C08974=1024.859,160.685,-112.460,168.492,47.875,158.974
C08975=1024.853,160.436,-112.438,168.489,47.879,158.974
C08976=1024.849,160.187,-112.416,168.486,47.884,158.975
C08977=1024.842,159.938,-112.393,168.482,47.888,158.975
C08978=1024.837,159.689,-112.372,168.480,47.892,158.976
C08979=1024.832,159.440,-112.349,168.476,47.897,158.976
C08980=1024.826,159.191,-112.328,168.472,47.901,158.977
C08981=1024.821,158.942,-112.306,168.470,47.905,158.977
C08982=1024.815,158.693,-112.285,168.466,47.910,158.978
C08983=1024.809,158.444,-112.263,168.464,47.914,158.978
C08984=1024.803,158.195,-112.241,168.460,47.918,158.978
C08985=1024.797,157.946,-112.220,168.456,47.923,158.979
C08986=1024.792,157.697,-112.198,168.454,47.928,158.979
C08987=1024.786,157.448,-112.177,168.450,47.932,158.980
C08988=1024.780,157.199,-112.155,168.446,47.937,158.980
C08989=1024.775,156.951,-112.134,168.444,47.941,158.981
C08990=1024.770,156.701,-112.112,168.440,47.946,158.981
C08991=1024.764,156.452,-112.091,168.438,47.950,158.982
C08992=1024.757,156.169,-112.066,168.433,47.955,158.982
C08993=1024.751,155.886,-112.042,168.430,47.960,158.983
C08994=1024.745,155.602,-112.017,168.426,47.965,158.983
C08995=1024.738,155.318,-111.992,168.423,47.970,158.984
C08996=1024.732,155.070,-111.971,168.419,47.974,158.984
C08997=1024.726,154.820,-111.950,168.416,47.979,158.985
C08998=1024.721,154.571,-111.929,168.414,47.984,158.985
C08999=1024.715,154.322,-111.907,168.410,47.988,158.985
C09000=1024.710,154.073,-111.885,168.407,47.992,158.986
C09001=1024.703,153.824,-111.864,168.404,47.997,158.986
C09002=1024.698,153.576,-111.843,168.401,48.001,158.987
C09003=1024.693,153.326,-111.822,168.397,48.006,158.987
C09004=1024.687,153.077,-111.800,168.394,48.010,158.988
C09005=1024.682,152.828,-111.779,168.391,48.015,158.988
C09006=1024.675,152.579,-111.757,168.388,48.019,158.989
C09007=1024.670,152.330,-111.736,168.385,48.023,158.989
C09008=1024.664,152.081,-111.715,168.382,48.028,158.990
C09009=1024.658,151.832,-111.693,168.378,48.033,158.990
C09010=1024.653,151.583,-111.673,168.375,48.037,158.990
C09011=1024.647,151.334,-111.651,168.372,48.042,158.991
C09012=1024.641,151.085,-111.630,168.369,48.046,158.992
C09013=1024.636,150.836,-111.609,168.366,48.051,158.992
C09014=1024.630,150.587,-111.588,168.363,48.055,158.992
C09015=1024.624,150.338,-111.566,168.360,48.059,158.993
C09016=1024.619,150.089,-111.546,168.356,48.064,158.993
C09017=1024.612,149.840,-111.524,168.354,48.069,158.994
C09018=1024.607,149.591,-111.503,168.350,48.073,158.994
C09019=1024.602,149.342,-111.482,168.347,48.077,158.995
C09020=1024.595,149.093,-111.460,168.344,48.082,158.995
C09021=1024.590,148.844,-111.440,168.341,48.087,158.996
C09022=1024.584,148.595,-111.418,168.338,48.091,158.996
C09023=1024.579,148.345,-111.398,168.335,48.095,158.997
C09024=1024.573,148.097,-111.376,168.332,48.100,158.997
C09025=1024.567,147.848,-111.355,168.329,48.105,158.998
C09026=1024.562,147.599,-111.334,168.325,48.109,158.998
C09027=1024.556,147.349,-111.313,168.322,48.113,158.998
C09028=1024.550,147.100,-111.292,168.319,48.118,158.999
C09029=1024.545,146.852,-111.271,168.316,48.123,158.999
C09030=1024.539,146.602,-111.250,168.313,48.127,159.000
C09031=1024.533,146.353,-111.229,168.310,48.131,159.000
C09032=1024.528,146.104,-111.208,168.307,48.136,159.001
C09033=1024.522,145.854,-111.187,168.304,48.141,159.001
C09034=1024.517,145.606,-111.166,168.301,48.145,159.002
C09035=1024.511,145.357,-111.145,168.298,48.150,159.002
C09036=1024.505,145.108,-111.124,168.295,48.155,159.003
C09037=1024.499,144.859,-111.104,168.291,48.159,159.003
C09038=1024.494,144.610,-111.083,168.289,48.163,159.004
C09039=1024.488,144.360,-111.062,168.285,48.168,159.004
C09040=1024.483,144.111,-111.041,168.282,48.173,159.005
C09041=1024.477,143.863,-111.021,168.280,48.177,159.005
C09042=1024.470,143.613,-110.999,168.276,48.182,159.006
C09043=1024.465,143.364,-110.979,168.274,48.187,159.006
C09044=1024.460,143.115,-110.958,168.270,48.191,159.006
C09045=1024.453,142.866,-110.937,168.267,48.195,159.007
C09046=1024.448,142.617,-110.917,168.264,48.200,159.008
C09047=1024.443,142.368,-110.896,168.261,48.205,159.008
C09048=1024.437,142.119,-110.875,168.258,48.209,159.009
C09049=1024.430,141.870,-110.855,168.255,48.214,159.009
C09050=1024.425,141.621,-110.834,168.252,48.219,159.010
C09051=1024.420,141.372,-110.813,168.249,48.222,159.010
C09052=1024.414,141.122,-110.792,168.246,48.227,159.010
C09053=1024.408,140.873,-110.771,168.243,48.232,159.011
C09054=1024.402,140.625,-110.751,168.240,48.237,159.011
C09055=1024.397,140.375,-110.731,168.237,48.241,159.012
C09056=1024.391,140.091,-110.707,168.234,48.246,159.012
C09057=1024.384,139.808,-110.683,168.231,48.251,159.013
C09058=1024.378,139.524,-110.659,168.226,48.257,159.013
C09059=1024.371,139.241,-110.636,168.223,48.262,159.014
C09060=1024.366,138.992,-110.616,168.221,48.267,159.015
C09061=1024.360,138.743,-110.595,168.217,48.271,159.015
C09062=1024.354,138.493,-110.574,168.214,48.275,159.015
C09063=1024.348,138.244,-110.554,168.211,48.280,159.016
C09064=1024.343,137.995,-110.534,168.208,48.285,159.017
C09065=1024.338,137.746,-110.513,168.205,48.289,159.017
C09066=1024.331,137.496,-110.493,168.202,48.294,159.018
C09067=1024.326,137.248,-110.471,168.199,48.299,159.018
C09068=1024.320,136.999,-110.451,168.197,48.303,159.019
C09069=1024.315,136.750,-110.431,168.193,48.308,159.019
C09070=1024.309,136.501,-110.410,168.191,48.313,159.020
C09071=1024.303,136.251,-110.390,168.188,48.316,159.020
C09072=1024.297,136.002,-110.369,168.184,48.321,159.020
C09073=1024.291,135.753,-110.349,168.182,48.326,159.021
C09074=1024.286,135.504,-110.329,168.178,48.331,159.021
C09075=1024.280,135.255,-110.309,168.176,48.335,159.022
C09076=1024.274,135.005,-110.288,168.173,48.340,159.022
C09077=1024.268,134.757,-110.268,168.170,48.345,159.023
C09078=1024.263,134.508,-110.248,168.167,48.349,159.023
C09079=1024.257,134.259,-110.228,168.164,48.354,159.024
C09080=1024.252,134.010,-110.207,168.161,48.359,159.024
C09081=1024.246,133.761,-110.187,168.158,48.363,159.025
C09082=1024.241,133.512,-110.167,168.155,48.368,159.025
C09083=1024.234,133.262,-110.147,168.152,48.373,159.026
C09084=1024.229,133.012,-110.126,168.149,48.377,159.026
C09085=1024.223,132.764,-110.106,168.146,48.382,159.027
C09086=1024.218,132.514,-110.086,168.143,48.386,159.027
C09087=1024.212,132.266,-110.066,168.140,48.391,159.028
C09088=1024.207,132.017,-110.045,168.138,48.395,159.028
C09089=1024.201,131.768,-110.025,168.134,48.400,159.029
C09090=1024.195,131.518,-110.004,168.132,48.405,159.029
C09091=1024.189,131.269,-109.984,168.128,48.409,159.030
C09092=1024.183,131.020,-109.964,168.126,48.414,159.030
C09093=1024.178,130.771,-109.945,168.123,48.419,159.031
C09094=1024.173,130.521,-109.924,168.120,48.423,159.031
C09095=1024.167,130.273,-109.904,168.117,48.428,159.032
C09096=1024.161,130.023,-109.884,168.114,48.433,159.032
C09097=1024.155,129.775,-109.864,168.112,48.437,159.033
C09098=1024.150,129.525,-109.844,168.108,48.442,159.033
C09099=1024.144,129.276,-109.824,168.105,48.447,159.034
C09100=1024.137,129.027,-109.804,168.102,48.452,159.034
C09101=1024.131,128.777,-109.785,168.099,48.456,159.035
C09102=1024.126,128.528,-109.764,168.097,48.461,159.035
C09103=1024.120,128.280,-109.744,168.094,48.465,159.036
C09104=1024.114,128.030,-109.725,168.091,48.470,159.036
C09105=1024.108,127.781,-109.705,168.088,48.475,159.037
C09106=1024.102,127.532,-109.685,168.085,48.480,159.037
C09107=1024.097,127.283,-109.666,168.083,48.485,159.038
C09108=1024.091,127.034,-109.646,168.079,48.490,159.039
C09109=1024.086,126.784,-109.626,168.077,48.494,159.039
C09110=1024.080,126.536,-109.606,168.073,48.499,159.040
C09111=1024.073,126.286,-109.586,168.071,48.504,159.040
C09112=1024.067,126.037,-109.567,168.067,48.509,159.041
C09113=1024.061,125.788,-109.547,168.065,48.513,159.041
C09114=1024.056,125.538,-109.527,168.062,48.518,159.042
C09115=1024.051,125.289,-109.507,168.059,48.523,159.042
C09116=1024.045,125.041,-109.487,168.056,48.527,159.043
C09117=1024.039,124.791,-109.468,168.053,48.532,159.043
C09118=1024.033,124.542,-109.448,168.050,48.537,159.044
C09119=1024.027,124.293,-109.428,168.047,48.541,159.044
C09120=1024.021,124.009,-109.406,168.044,48.547,159.045
C09121=1024.014,123.726,-109.384,168.041,48.552,159.046
C09122=1024.008,123.442,-109.361,168.038,48.557,159.046
C09123=1024.002,123.158,-109.339,168.035,48.563,159.047
C09124=1023.996,122.909,-109.319,168.031,48.568,159.047
C09125=1023.990,122.660,-109.299,168.029,48.572,159.048
C09126=1023.984,122.411,-109.279,168.026,48.577,159.048
C09127=1023.978,122.161,-109.260,168.023,48.582,159.049
C09128=1023.972,121.913,-109.240,168.020,48.586,159.049
C09129=1023.967,121.663,-109.221,168.017,48.591,159.050
C09130=1023.961,121.414,-109.200,168.014,48.596,159.050
C09131=1023.956,121.165,-109.181,168.012,48.600,159.051
C09132=1023.950,120.916,-109.161,168.009,48.605,159.051
C09133=1023.944,120.666,-109.142,168.006,48.610,159.052
C09134=1023.938,120.417,-109.123,168.003,48.614,159.052
C09135=1023.932,120.168,-109.103,168.000,48.619,159.053
C09136=1023.927,119.919,-109.084,167.998,48.624,159.053
C09137=1023.921,119.670,-109.063,167.994,48.629,159.054
C09138=1023.916,119.420,-109.044,167.992,48.633,159.054
C09139=1023.910,119.171,-109.024,167.989,48.638,159.055
C09140=1023.904,118.922,-109.005,167.986,48.643,159.055
C09141=1023.898,118.672,-108.985,167.984,48.647,159.056
C09142=1023.892,118.424,-108.965,167.980,48.652,159.056
C09143=1023.887,118.175,-108.946,167.978,48.657,159.057
C09144=1023.882,117.926,-108.927,167.976,48.661,159.057
C09145=1023.876,117.676,-108.907,167.972,48.666,159.058
C09146=1023.871,117.427,-108.887,167.970,48.671,159.058
C09147=1023.865,117.178,-108.867,167.966,48.675,159.059
C09148=1023.859,116.929,-108.848,167.964,48.680,159.059
C09149=1023.853,116.679,-108.829,167.961,48.685,159.060
C09150=1023.847,116.430,-108.809,167.958,48.689,159.060
C09151=1023.842,116.182,-108.790,167.956,48.694,159.061
C09152=1023.837,115.932,-108.771,167.953,48.699,159.062
C09153=1023.831,115.683,-108.750,167.950,48.703,159.062
C09154=1023.826,115.434,-108.731,167.947,48.708,159.063
C09155=1023.820,115.184,-108.712,167.945,48.713,159.063
C09156=1023.814,114.935,-108.693,167.941,48.718,159.064
C09157=1023.808,114.686,-108.673,167.939,48.722,159.064
C09158=1023.803,114.437,-108.654,167.936,48.726,159.064
C09159=1023.797,114.188,-108.635,167.933,48.731,159.065
C09160=1023.791,113.939,-108.615,167.930,48.735,159.065
C09161=1023.786,113.690,-108.595,167.928,48.740,159.066
C09162=1023.781,113.440,-108.575,167.925,48.745,159.066
C09163=1023.775,113.190,-108.556,167.922,48.750,159.067
C09164=1023.770,112.942,-108.537,167.920,48.754,159.067
C09165=1023.764,112.693,-108.517,167.917,48.759,159.068
C09166=1023.758,112.443,-108.498,167.914,48.764,159.068
C09167=1023.753,112.194,-108.479,167.912,48.768,159.069
C09168=1023.746,111.945,-108.460,167.908,48.773,159.069
C09169=1023.741,111.695,-108.441,167.906,48.778,159.070
C09170=1023.735,111.447,-108.422,167.903,48.782,159.071
C09171=1023.730,111.197,-108.403,167.900,48.787,159.071
C09172=1023.724,110.948,-108.384,167.897,48.792,159.072
C09173=1023.718,110.698,-108.364,167.895,48.796,159.072
C09174=1023.712,110.450,-108.345,167.892,48.801,159.073
C09175=1023.707,110.201,-108.326,167.889,48.806,159.073
C09176=1023.701,109.952,-108.307,167.886,48.811,159.074
C09177=1023.695,109.702,-108.288,167.884,48.816,159.074
C09178=1023.689,109.453,-108.268,167.881,48.821,159.075
C09179=1023.683,109.204,-108.250,167.878,48.825,159.075
C09180=1023.678,108.954,-108.231,167.876,48.830,159.076
C09181=1023.673,108.705,-108.212,167.873,48.835,159.076
C09182=1023.666,108.456,-108.194,167.870,48.840,159.077
C09183=1023.660,108.206,-108.175,167.867,48.844,159.077
C09184=1023.653,107.923,-108.153,167.864,48.850,159.078
C09185=1023.647,107.639,-108.131,167.861,48.855,159.079
C09186=1023.641,107.355,-108.110,167.858,48.861,159.079
C09187=1023.634,107.071,-108.089,167.855,48.866,159.080
C09188=1023.629,106.822,-108.070,167.852,48.871,159.080
C09189=1023.622,106.573,-108.051,167.849,48.876,159.081
C09190=1023.617,106.323,-108.032,167.847,48.881,159.081
C09191=1023.611,106.074,-108.013,167.843,48.885,159.082
C09192=1023.605,105.825,-107.994,167.841,48.890,159.082
C09193=1023.599,105.576,-107.975,167.839,48.895,159.083
C09194=1023.594,105.327,-107.956,167.835,48.900,159.083
C09195=1023.588,105.078,-107.938,167.833,48.904,159.084
C09196=1023.582,104.828,-107.919,167.830,48.910,159.085
C09197=1023.577,104.579,-107.900,167.827,48.914,159.085
C09198=1023.570,104.330,-107.881,167.825,48.919,159.086
C09199=1023.565,104.081,-107.862,167.821,48.924,159.086
C09200=1023.559,103.832,-107.844,167.819,48.928,159.087
C09201=1023.553,103.582,-107.825,167.817,48.933,159.087
C09202=1023.548,103.333,-107.806,167.813,48.938,159.088
C09203=1023.542,103.084,-107.787,167.811,48.943,159.088
C09204=1023.536,102.834,-107.768,167.809,48.947,159.089
C09205=1023.531,102.585,-107.749,167.805,48.952,159.089
C09206=1023.525,102.336,-107.731,167.803,48.957,159.090
C09207=1023.519,102.086,-107.712,167.800,48.961,159.090
C09208=1023.513,101.837,-107.694,167.797,48.966,159.091
C09209=1023.508,101.589,-107.675,167.795,48.971,159.091
C09210=1023.502,101.339,-107.656,167.792,48.976,159.092
C09211=1023.496,101.089,-107.637,167.790,48.980,159.092
C09212=1023.491,100.841,-107.619,167.786,48.985,159.093
C09213=1023.485,100.591,-107.599,167.784,48.990,159.093
C09214=1023.480,100.342,-107.582,167.782,48.994,159.094
C09215=1023.474,100.093,-107.563,167.778,48.999,159.094
C09216=1023.468,99.844,-107.544,167.776,49.004,159.095
C09217=1023.462,99.594,-107.525,167.773,49.008,159.095
C09218=1023.457,99.345,-107.507,167.770,49.014,159.096
C09219=1023.451,99.096,-107.488,167.768,49.019,159.097
C09220=1023.445,98.847,-107.470,167.766,49.023,159.097
C09221=1023.440,98.597,-107.451,167.762,49.028,159.098
C09222=1023.433,98.348,-107.433,167.760,49.033,159.098
C09223=1023.428,98.099,-107.415,167.756,49.038,159.099
C09224=1023.422,97.849,-107.396,167.754,49.043,159.099
C09225=1023.416,97.600,-107.378,167.752,49.048,159.100
C09226=1023.410,97.352,-107.359,167.749,49.053,159.100
C09227=1023.405,97.102,-107.341,167.746,49.057,159.101
C09228=1023.398,96.852,-107.322,167.744,49.062,159.101
C09229=1023.393,96.603,-107.305,167.740,49.067,159.102
C09230=1023.387,96.354,-107.285,167.738,49.071,159.102
C09231=1023.381,96.105,-107.268,167.736,49.077,159.103
C09232=1023.375,95.856,-107.249,167.733,49.082,159.104
C09233=1023.370,95.606,-107.231,167.730,49.086,159.104
C09234=1023.364,95.357,-107.212,167.728,49.091,159.105
C09235=1023.358,95.108,-107.194,167.724,49.096,159.105
C09236=1023.353,94.859,-107.176,167.722,49.100,159.106
C09237=1023.346,94.609,-107.158,167.720,49.105,159.106
C09238=1023.340,94.360,-107.139,167.716,49.110,159.107
C09239=1023.335,94.111,-107.121,167.714,49.115,159.107
C09240=1023.329,93.861,-107.103,167.712,49.120,159.108
C09241=1023.323,93.612,-107.085,167.709,49.125,159.108
C09242=1023.318,93.362,-107.066,167.706,49.130,159.109
C09243=1023.312,93.114,-107.048,167.704,49.134,159.109
C09244=1023.306,92.864,-107.030,167.700,49.139,159.110
C09245=1023.301,92.616,-107.011,167.698,49.144,159.110
C09246=1023.295,92.366,-106.993,167.696,49.148,159.111
C09247=1023.289,92.116,-106.975,167.692,49.153,159.111
C09248=1023.282,91.833,-106.954,167.690,49.159,159.112
C09249=1023.276,91.548,-106.933,167.687,49.164,159.113
C09250=1023.270,91.265,-106.912,167.684,49.169,159.113
C09251=1023.263,90.981,-106.892,167.681,49.175,159.114
C09252=1023.257,90.732,-106.874,167.678,49.179,159.114
C09253=1023.252,90.482,-106.855,167.675,49.184,159.115
C09254=1023.246,90.234,-106.837,167.673,49.189,159.115
C09255=1023.240,89.984,-106.819,167.670,49.194,159.116
C09256=1023.235,89.735,-106.801,167.667,49.199,159.116
C09257=1023.229,89.486,-106.782,167.664,49.203,159.117
C09258=1023.223,89.236,-106.764,167.662,49.208,159.117
C09259=1023.217,88.987,-106.747,167.659,49.214,159.118
C09260=1023.211,88.738,-106.729,167.657,49.218,159.118
C09261=1023.205,88.488,-106.711,167.654,49.223,159.119
C09262=1023.199,88.240,-106.693,167.651,49.228,159.119
C09263=1023.193,87.990,-106.675,167.649,49.232,159.120
C09264=1023.188,87.741,-106.657,167.647,49.238,159.121
C09265=1023.182,87.491,-106.639,167.643,49.243,159.121
C09266=1023.176,87.242,-106.622,167.641,49.247,159.122
C09267=1023.170,86.992,-106.604,167.638,49.252,159.122
C09268=1023.164,86.744,-106.586,167.635,49.257,159.123
C09269=1023.158,86.494,-106.568,167.633,49.262,159.123
C09270=1023.153,86.245,-106.550,167.631,49.267,159.124
C09271=1023.147,85.995,-106.532,167.627,49.272,159.124
C09272=1023.141,85.746,-106.515,167.625,49.277,159.125
C09273=1023.135,85.497,-106.497,167.623,49.281,159.125
C09274=1023.129,85.247,-106.479,167.619,49.286,159.126
C09275=1023.123,84.998,-106.461,167.617,49.291,159.126
C09276=1023.117,84.749,-106.443,167.615,49.296,159.127
C09277=1023.111,84.500,-106.425,167.612,49.301,159.128
C09278=1023.106,84.251,-106.407,167.609,49.306,159.128
C09279=1023.100,84.002,-106.390,167.607,49.310,159.129
C09280=1023.094,83.752,-106.372,167.603,49.315,159.129
C09281=1023.089,83.503,-106.354,167.601,49.320,159.130
C09282=1023.083,83.253,-106.336,167.599,49.325,159.130
C09283=1023.077,83.004,-106.319,167.595,49.330,159.131
C09284=1023.072,82.754,-106.300,167.593,49.335,159.131
C09285=1023.066,82.505,-106.283,167.591,49.340,159.132
C09286=1023.061,82.256,-106.265,167.588,49.345,159.132
C09287=1023.054,82.006,-106.247,167.585,49.349,159.133
C09288=1023.049,81.757,-106.230,167.583,49.354,159.133
C09289=1023.043,81.507,-106.212,167.580,49.359,159.134
C09290=1023.037,81.258,-106.194,167.577,49.364,159.134
C09291=1023.032,81.009,-106.177,167.575,49.368,159.135
C09292=1023.026,80.759,-106.159,167.573,49.373,159.135
C09293=1023.020,80.510,-106.141,167.569,49.378,159.136
C09294=1023.015,80.261,-106.123,167.567,49.382,159.136
C09295=1023.008,80.012,-106.106,167.564,49.387,159.137
C09296=1023.002,79.763,-106.089,167.561,49.392,159.137
C09297=1022.997,79.514,-106.071,167.559,49.397,159.138
C09298=1022.991,79.264,-106.053,167.557,49.402,159.139
C09299=1022.985,79.015,-106.036,167.554,49.407,159.139
C09300=1022.979,78.765,-106.018,167.551,49.412,159.140
C09301=1022.973,78.516,-106.000,167.549,49.416,159.140
C09302=1022.968,78.267,-105.982,167.546,49.421,159.141
C09303=1022.962,78.018,-105.965,167.543,49.426,159.141
C09304=1022.956,77.768,-105.947,167.541,49.431,159.142
C09305=1022.951,77.519,-105.929,167.538,49.435,159.142
C09306=1022.945,77.270,-105.911,167.536,49.440,159.143
C09307=1022.939,77.020,-105.895,167.533,49.445,159.143
C09308=1022.934,76.771,-105.877,167.530,49.450,159.144
C09309=1022.928,76.521,-105.859,167.528,49.454,159.144
C09310=1022.922,76.272,-105.842,167.525,49.459,159.145
C09311=1022.916,76.023,-105.825,167.522,49.464,159.145
C09312=1022.909,75.739,-105.804,167.519,49.470,159.146
C09313=1022.903,75.455,-105.785,167.516,49.475,159.146
C09314=1022.896,75.171,-105.765,167.513,49.481,159.147
C09315=1022.890,74.888,-105.746,167.510,49.487,159.148
C09316=1022.884,74.638,-105.728,167.508,49.491,159.148
C09317=1022.878,74.388,-105.711,167.505,49.496,159.149
C09318=1022.872,74.140,-105.694,167.502,49.501,159.149
C09319=1022.867,73.891,-105.676,167.500,49.506,159.150
C09320=1022.860,73.641,-105.658,167.498,49.511,159.151
C09321=1022.854,73.392,-105.642,167.494,49.516,159.151
C09322=1022.849,73.143,-105.625,167.492,49.521,159.151
C09323=1022.843,72.893,-105.607,167.490,49.525,159.152
C09324=1022.837,72.644,-105.590,167.486,49.530,159.152
C09325=1022.831,72.394,-105.573,167.484,49.535,159.153
C09326=1022.826,72.145,-105.555,167.482,49.540,159.154
C09327=1022.820,71.895,-105.538,167.479,49.544,159.154
C09328=1022.814,71.646,-105.521,167.476,49.549,159.154
C09329=1022.808,71.397,-105.503,167.474,49.554,159.155
C09330=1022.803,71.148,-105.487,167.472,49.560,159.156
C09331=1022.796,70.898,-105.469,167.468,49.565,159.156
C09332=1022.791,70.649,-105.452,167.466,49.569,159.157
C09333=1022.785,70.400,-105.435,167.464,49.574,159.157
C09334=1022.779,70.151,-105.418,167.460,49.579,159.158
C09335=1022.773,69.900,-105.401,167.458,49.584,159.158
C09336=1022.768,69.651,-105.383,167.456,49.588,159.159
C09337=1022.762,69.403,-105.366,167.453,49.593,159.159
C09338=1022.756,69.153,-105.349,167.450,49.598,159.160
C09339=1022.750,68.903,-105.331,167.448,49.603,159.160
C09340=1022.744,68.654,-105.315,167.445,49.607,159.161
C09341=1022.739,68.405,-105.298,167.442,49.612,159.161
C09342=1022.733,68.156,-105.281,167.440,49.617,159.162
C09343=1022.727,67.906,-105.264,167.438,49.622,159.162
C09344=1022.722,67.656,-105.247,167.434,49.627,159.163
C09345=1022.715,67.407,-105.230,167.432,49.632,159.163
C09346=1022.710,67.158,-105.213,167.430,49.637,159.164
C09347=1022.704,66.909,-105.196,167.426,49.642,159.164
C09348=1022.699,66.659,-105.179,167.424,49.646,159.165
C09349=1022.692,66.410,-105.162,167.422,49.651,159.165
C09350=1022.686,66.160,-105.145,167.419,49.656,159.166
C09351=1022.680,65.912,-105.128,167.416,49.661,159.166
C09352=1022.675,65.662,-105.111,167.414,49.666,159.167
C09353=1022.669,65.413,-105.095,167.412,49.671,159.168
C09354=1022.663,65.163,-105.077,167.409,49.676,159.168
C09355=1022.657,64.913,-105.060,167.406,49.681,159.169
C09356=1022.651,64.664,-105.043,167.404,49.685,159.169
C09357=1022.646,64.415,-105.027,167.401,49.690,159.170
C09358=1022.640,64.166,-105.010,167.398,49.695,159.170
C09359=1022.634,63.917,-104.993,167.396,49.700,159.171
C09360=1022.628,63.667,-104.976,167.393,49.705,159.171
C09361=1022.622,63.418,-104.959,167.390,49.709,159.172
C09362=1022.616,63.168,-104.942,167.388,49.715,159.172
C09363=1022.611,62.919,-104.925,167.385,49.720,159.173
C09364=1022.605,62.669,-104.909,167.383,49.725,159.173
C09365=1022.598,62.420,-104.892,167.380,49.729,159.174
C09366=1022.592,62.170,-104.876,167.377,49.735,159.174
C09367=1022.586,61.921,-104.859,167.375,49.740,159.175
C09368=1022.580,61.672,-104.843,167.372,49.745,159.175
C09369=1022.575,61.422,-104.826,167.369,49.749,159.176
C09370=1022.569,61.173,-104.809,167.367,49.754,159.177
C09371=1022.563,60.924,-104.793,167.364,49.760,159.177
C09372=1022.556,60.674,-104.776,167.362,49.765,159.178
C09373=1022.550,60.425,-104.760,167.358,49.770,159.178
C09374=1022.544,60.175,-104.744,167.356,49.774,159.179
C09375=1022.539,59.926,-104.727,167.354,49.780,159.179
C09376=1022.532,59.642,-104.708,167.351,49.785,159.180
C09377=1022.525,59.358,-104.690,167.348,49.790,159.180
C09378=1022.519,59.074,-104.671,167.345,49.796,159.181
C09379=1022.512,58.790,-104.652,167.342,49.802,159.182
C09380=1022.506,58.541,-104.635,167.339,49.807,159.182
C09381=1022.500,58.292,-104.619,167.337,49.812,159.183
C09382=1022.494,58.042,-104.603,167.334,49.817,159.183
C09383=1022.488,57.792,-104.586,167.331,49.822,159.184
C09384=1022.482,57.543,-104.569,167.329,49.827,159.184
C09385=1022.476,57.293,-104.553,167.326,49.831,159.185
C09386=1022.470,57.045,-104.536,167.323,49.836,159.185
C09387=1022.464,56.795,-104.520,167.321,49.842,159.186
C09388=1022.458,56.546,-104.504,167.319,49.847,159.186
C09389=1022.452,56.296,-104.487,167.316,49.852,159.187
C09390=1022.447,56.047,-104.471,167.313,49.856,159.187
C09391=1022.441,55.797,-104.454,167.311,49.861,159.188
C09392=1022.435,55.548,-104.438,167.308,49.866,159.188
C09393=1022.429,55.299,-104.422,167.305,49.871,159.189
C09394=1022.423,55.049,-104.406,167.303,49.876,159.189
C09395=1022.417,54.800,-104.389,167.300,49.881,159.190
C09396=1022.412,54.550,-104.372,167.298,49.886,159.191
C09397=1022.406,54.301,-104.356,167.294,49.891,159.191
C09398=1022.400,54.052,-104.340,167.292,49.896,159.192
C09399=1022.394,53.802,-104.324,167.290,49.900,159.192
C09400=1022.388,53.553,-104.307,167.288,49.905,159.193
C09401=1022.382,53.304,-104.291,167.284,49.910,159.193
C09402=1022.376,53.054,-104.275,167.282,49.915,159.194
C09403=1022.371,52.805,-104.258,167.280,49.920,159.194
C09404=1022.365,52.555,-104.242,167.276,49.925,159.195
C09405=1022.359,52.306,-104.226,167.274,49.929,159.195
C09406=1022.353,52.057,-104.209,167.272,49.934,159.196
C09407=1022.347,51.807,-104.193,167.268,49.939,159.196
C09408=1022.341,51.558,-104.177,167.266,49.944,159.197
C09409=1022.335,51.309,-104.161,167.264,49.949,159.197
C09410=1022.329,51.059,-104.144,167.261,49.954,159.198
C09411=1022.324,50.810,-104.127,167.259,49.959,159.198
C09412=1022.318,50.560,-104.111,167.256,49.964,159.199
C09413=1022.312,50.311,-104.095,167.253,49.969,159.199
C09414=1022.306,50.062,-104.079,167.251,49.974,159.200
C09415=1022.301,49.812,-104.063,167.248,49.978,159.200
C09416=1022.295,49.562,-104.047,167.245,49.983,159.201
C09417=1022.289,49.313,-104.031,167.243,49.988,159.201
C09418=1022.283,49.064,-104.014,167.240,49.993,159.202
C09419=1022.277,48.814,-103.998,167.238,49.998,159.202
C09420=1022.272,48.565,-103.982,167.235,50.003,159.203
C09421=1022.266,48.316,-103.965,167.233,50.007,159.203
C09422=1022.260,48.067,-103.949,167.230,50.012,159.204
C09423=1022.254,47.817,-103.933,167.227,50.017,159.204
C09424=1022.249,47.567,-103.917,167.224,50.021,159.204
C09425=1022.243,47.318,-103.901,167.222,50.026,159.205
C09426=1022.237,47.068,-103.885,167.220,50.031,159.206
C09427=1022.232,46.819,-103.868,167.216,50.036,159.206
C09428=1022.226,46.569,-103.852,167.214,50.040,159.206
C09429=1022.220,46.320,-103.835,167.212,50.045,159.207
C09430=1022.215,46.071,-103.820,167.209,50.050,159.207
C09431=1022.209,45.822,-103.804,167.206,50.055,159.208
C09432=1022.203,45.572,-103.788,167.204,50.060,159.208
C09433=1022.197,45.323,-103.771,167.202,50.064,159.209
C09434=1022.191,45.073,-103.755,167.198,50.070,159.209
C09435=1022.186,44.823,-103.739,167.196,50.074,159.210
C09436=1022.180,44.574,-103.723,167.194,50.079,159.211
C09437=1022.175,44.325,-103.707,167.191,50.083,159.211
C09438=1022.169,44.076,-103.691,167.188,50.088,159.211
C09439=1022.163,43.826,-103.675,167.186,50.093,159.212
C09440=1022.156,43.542,-103.657,167.183,50.099,159.212
C09441=1022.150,43.258,-103.638,167.179,50.104,159.213
C09442=1022.143,42.974,-103.620,167.177,50.109,159.214
C09443=1022.136,42.689,-103.601,167.174,50.114,159.214
C09444=1022.131,42.440,-103.586,167.171,50.119,159.214
C09445=1022.125,42.191,-103.570,167.169,50.124,159.215
C09446=1022.120,41.941,-103.554,167.166,50.129,159.215
C09447=1022.114,41.692,-103.538,167.163,50.134,159.216
C09448=1022.108,41.442,-103.522,167.161,50.139,159.216
C09449=1022.101,41.192,-103.507,167.158,50.143,159.217
C09450=1022.096,40.944,-103.491,167.155,50.148,159.217
C09451=1022.090,40.694,-103.475,167.153,50.153,159.218
C09452=1022.084,40.445,-103.459,167.151,50.158,159.218
C09453=1022.079,40.195,-103.444,167.147,50.163,159.219
C09454=1022.073,39.945,-103.427,167.145,50.168,159.219
C09455=1022.067,39.697,-103.412,167.143,50.172,159.220
C09456=1022.061,39.447,-103.396,167.139,50.178,159.220
C09457=1022.055,39.198,-103.380,167.137,50.182,159.221
C09458=1022.049,38.948,-103.365,167.135,50.187,159.221
C09459=1022.043,38.698,-103.348,167.133,50.192,159.222
C09460=1022.038,38.449,-103.333,167.129,50.197,159.222
C09461=1022.032,38.200,-103.318,167.127,50.202,159.223
C09462=1022.026,37.950,-103.302,167.125,50.206,159.223
C09463=1022.020,37.701,-103.286,167.122,50.211,159.224
C09464=1022.015,37.451,-103.271,167.119,50.216,159.224
C09465=1022.009,37.202,-103.254,167.117,50.221,159.225
C09466=1022.003,36.952,-103.239,167.114,50.226,159.225
C09467=1021.997,36.702,-103.224,167.111,50.231,159.226
C09468=1021.991,36.453,-103.208,167.109,50.236,159.226
C09469=1021.985,36.204,-103.193,167.106,50.241,159.227
C09470=1021.979,35.955,-103.177,167.104,50.245,159.227
C09471=1021.974,35.705,-103.161,167.101,50.250,159.228
C09472=1021.967,35.455,-103.146,167.098,50.255,159.228
C09473=1021.962,35.206,-103.130,167.096,50.260,159.229
C09474=1021.956,34.957,-103.115,167.093,50.265,159.229
C09475=1021.950,34.707,-103.100,167.090,50.270,159.230
C09476=1021.944,34.457,-103.084,167.088,50.275,159.230
C09477=1021.938,34.209,-103.069,167.085,50.280,159.231
C09478=1021.933,33.959,-103.054,167.082,50.285,159.231
C09479=1021.926,33.709,-103.039,167.080,50.289,159.232
C09480=1021.921,33.460,-103.023,167.077,50.294,159.232
C09481=1021.915,33.211,-103.008,167.075,50.299,159.233
C09482=1021.909,32.961,-102.992,167.071,50.304,159.233
C09483=1021.903,32.711,-102.976,167.069,50.309,159.233
C09484=1021.897,32.462,-102.961,167.067,50.314,159.234
C09485=1021.892,32.212,-102.946,167.064,50.319,159.234
C09486=1021.885,31.963,-102.931,167.061,50.324,159.235
C09487=1021.880,31.714,-102.915,167.059,50.328,159.235
C09488=1021.873,31.464,-102.900,167.056,50.333,159.236
C09489=1021.868,31.214,-102.885,167.053,50.338,159.236
C09490=1021.863,30.965,-102.869,167.051,50.343,159.237
C09491=1021.856,30.716,-102.854,167.048,50.348,159.237
C09492=1021.850,30.466,-102.838,167.046,50.353,159.238
C09493=1021.845,30.217,-102.824,167.043,50.358,159.238
C09494=1021.839,29.967,-102.808,167.040,50.363,159.239
C09495=1021.833,29.718,-102.793,167.038,50.368,159.239
C09496=1021.828,29.468,-102.778,167.036,50.372,159.240
C09497=1021.821,29.219,-102.762,167.032,50.377,159.240
C09498=1021.816,28.970,-102.747,167.030,50.382,159.241
C09499=1021.810,28.720,-102.732,167.028,50.387,159.241
C09500=1021.804,28.470,-102.717,167.025,50.392,159.242
C09501=1021.799,28.221,-102.701,167.022,50.396,159.242
C09502=1021.792,27.971,-102.686,167.020,50.401,159.243
C09503=1021.786,27.722,-102.670,167.016,50.406,159.243
C09504=1021.777,27.319,-102.647,167.012,50.414,159.244
C09505=1021.768,26.917,-102.622,167.008,50.422,159.245
C09506=1021.758,26.513,-102.598,167.004,50.430,159.245
C09507=1021.748,26.111,-102.574,167.000,50.437,159.246
C09508=1021.743,25.861,-102.558,166.997,50.442,159.247
C09509=1021.737,25.612,-102.543,166.994,50.447,159.247
C09510=1021.731,25.362,-102.528,166.992,50.452,159.248
C09511=1021.725,25.113,-102.513,166.989,50.457,159.248
C09512=1021.719,24.864,-102.498,166.986,50.462,159.248
C09513=1021.713,24.614,-102.483,166.984,50.467,159.249
C09514=1021.708,24.365,-102.468,166.981,50.472,159.249
C09515=1021.701,24.115,-102.453,166.979,50.477,159.250
C09516=1021.693,23.735,-102.431,166.974,50.485,159.251
C09517=1021.684,23.354,-102.409,166.970,50.492,159.251
C09518=1021.674,22.974,-102.385,166.967,50.499,159.252
C09519=1021.666,22.594,-102.363,166.962,50.506,159.253
C09520=1021.660,22.344,-102.348,166.960,50.511,159.253
C09521=1021.654,22.095,-102.333,166.957,50.516,159.254
C09522=1021.648,21.845,-102.318,166.954,50.521,159.254
C09523=1021.642,21.596,-102.303,166.952,50.526,159.255
C09524=1021.637,21.346,-102.288,166.949,50.531,159.255
C09525=1021.631,21.097,-102.274,166.947,50.536,159.256
C09526=1021.625,20.847,-102.259,166.943,50.541,159.256
C09527=1021.620,20.598,-102.244,166.941,50.546,159.257
C09528=1021.613,20.348,-102.229,166.939,50.550,159.257
C09529=1021.608,20.099,-102.214,166.936,50.556,159.258
C09530=1021.602,19.849,-102.199,166.933,50.560,159.258
C09531=1021.596,19.600,-102.184,166.931,50.564,159.258
C09532=1021.590,19.350,-102.170,166.927,50.570,159.259
C09533=1021.584,19.101,-102.155,166.925,50.574,159.259
C09534=1021.579,18.851,-102.140,166.923,50.579,159.260
C09535=1021.573,18.602,-102.125,166.920,50.584,159.260
C09536=1021.567,18.352,-102.111,166.917,50.589,159.261
C09537=1021.561,18.103,-102.096,166.914,50.594,159.261
C09538=1021.555,17.853,-102.081,166.912,50.599,159.262
C09539=1021.549,17.604,-102.067,166.910,50.604,159.262
C09540=1021.543,17.354,-102.053,166.907,50.609,159.263
C09541=1021.538,17.105,-102.037,166.904,50.614,159.263
C09542=1021.531,16.855,-102.022,166.901,50.618,159.263
C09543=1021.526,16.605,-102.009,166.898,50.623,159.264
C09544=1021.520,16.356,-101.994,166.896,50.628,159.264
C09545=1021.514,16.107,-101.979,166.893,50.633,159.265
C09546=1021.508,15.857,-101.965,166.891,50.638,159.265
C09547=1021.503,15.607,-101.950,166.887,50.643,159.266
C09548=1021.497,15.358,-101.935,166.885,50.648,159.266
C09549=1021.491,15.108,-101.921,166.883,50.653,159.267
C09550=1021.485,14.859,-101.906,166.880,50.658,159.267
C09551=1021.479,14.609,-101.891,166.877,50.662,159.267
C09552=1021.473,14.360,-101.877,166.874,50.667,159.268
C09553=1021.467,14.111,-101.863,166.872,50.672,159.268
C09554=1021.462,13.861,-101.847,166.869,50.677,159.269
C09555=1021.456,13.611,-101.833,166.866,50.682,159.269
C09556=1021.450,13.362,-101.818,166.864,50.686,159.270
C09557=1021.444,13.112,-101.805,166.861,50.692,159.270
C09558=1021.439,12.863,-101.790,166.858,50.696,159.271
C09559=1021.432,12.613,-101.776,166.855,50.702,159.271
C09560=1021.426,12.364,-101.762,166.853,50.706,159.272
C09561=1021.420,12.114,-101.748,166.851,50.711,159.272
C09562=1021.414,11.865,-101.733,166.848,50.716,159.273
C09563=1021.409,11.615,-101.719,166.845,50.721,159.273
C09564=1021.402,11.332,-101.703,166.842,50.726,159.274
C09565=1021.395,11.050,-101.686,166.838,50.732,159.274
C09566=1021.388,10.767,-101.670,166.835,50.738,159.275
C09567=1021.381,10.485,-101.655,166.832,50.743,159.275
C09568=1021.375,10.234,-101.641,166.830,50.748,159.276
C09569=1021.369,9.985,-101.626,166.827,50.753,159.276
C09570=1021.364,9.736,-101.612,166.824,50.758,159.276
C09571=1021.358,9.486,-101.598,166.822,50.763,159.277
C09572=1021.352,9.237,-101.583,166.819,50.768,159.277
C09573=1021.346,8.987,-101.569,166.817,50.773,159.278
C09574=1021.340,8.737,-101.554,166.813,50.778,159.278
C09575=1021.334,8.488,-101.541,166.811,50.783,159.279
C09576=1021.328,8.239,-101.527,166.808,50.788,159.279
C09577=1021.322,7.989,-101.512,166.806,50.793,159.280
C09578=1021.316,7.739,-101.498,166.802,50.797,159.280
C09579=1021.311,7.490,-101.485,166.800,50.802,159.281
C09580=1021.305,7.241,-101.470,166.798,50.807,159.281
C09581=1021.298,6.991,-101.456,166.795,50.812,159.281
C09582=1021.293,6.741,-101.443,166.792,50.817,159.282
C09583=1021.287,6.492,-101.428,166.789,50.822,159.282
C09584=1021.281,6.242,-101.414,166.787,50.827,159.283
C09585=1021.276,5.992,-101.400,166.784,50.832,159.283
C09586=1021.270,5.743,-101.385,166.781,50.836,159.284
C09587=1021.264,5.494,-101.371,166.778,50.841,159.284
C09588=1021.258,5.244,-101.358,166.776,50.846,159.284
C09589=1021.252,4.994,-101.344,166.773,50.851,159.285
C09590=1021.246,4.745,-101.329,166.770,50.856,159.285
C09591=1021.241,4.496,-101.315,166.768,50.861,159.286
C09592=1021.235,4.246,-101.301,166.764,50.866,159.286
C09593=1021.229,3.997,-101.287,166.762,50.870,159.287
C09594=1021.223,3.747,-101.273,166.759,50.876,159.287
C09595=1021.217,3.498,-101.260,166.757,50.880,159.288
C09596=1021.211,3.247,-101.245,166.754,50.885,159.288
C09597=1021.206,2.998,-101.231,166.751,50.890,159.288
C09598=1021.200,2.749,-101.217,166.749,50.894,159.289
C09599=1021.194,2.499,-101.203,166.745,50.900,159.289
C09600=1021.188,2.249,-101.189,166.743,50.904,159.290
C09601=1021.182,2.000,-101.176,166.741,50.909,159.290
C09602=1021.177,1.750,-101.162,166.737,50.914,159.290
C09603=1021.171,1.501,-101.147,166.735,50.919,159.291
C09604=1021.165,1.252,-101.133,166.732,50.924,159.291
C09605=1021.160,1.002,-101.119,166.730,50.929,159.292
C09606=1021.153,0.752,-101.106,166.727,50.933,159.292
C09607=1021.148,0.503,-101.092,166.724,50.938,159.293
C09608=1021.142,0.253,-101.078,166.722,50.943,159.293
C09609=1021.136,0.004,-101.063,166.718,50.947,159.293
C09610=1021.131,-0.246,-101.050,166.716,50.952,159.294
C09611=1021.125,-0.495,-101.036,166.714,50.957,159.294
C09612=1021.119,-0.745,-101.022,166.710,50.962,159.295
C09613=1021.113,-0.995,-101.008,166.708,50.966,159.295
C09614=1021.108,-1.244,-100.994,166.705,50.971,159.295
C09615=1021.102,-1.494,-100.980,166.702,50.976,159.296
C09616=1021.097,-1.743,-100.967,166.700,50.980,159.296
C09617=1021.091,-1.993,-100.953,166.697,50.986,159.297
C09618=1021.085,-2.242,-100.939,166.694,50.990,159.297
C09619=1021.079,-2.492,-100.924,166.691,50.995,159.297
C09620=1021.073,-2.741,-100.911,166.689,51.000,159.298
C09621=1021.068,-2.991,-100.897,166.686,51.005,159.298
C09622=1021.062,-3.241,-100.883,166.683,51.009,159.299
C09623=1021.056,-3.490,-100.870,166.681,51.014,159.299
C09624=1021.050,-3.739,-100.856,166.677,51.019,159.300
C09625=1021.045,-3.989,-100.842,166.675,51.023,159.300
C09626=1021.040,-4.239,-100.828,166.673,51.028,159.300
C09627=1021.033,-4.489,-100.814,166.669,51.033,159.301
C09628=1021.027,-4.770,-100.800,166.666,51.038,159.301
C09629=1021.020,-5.050,-100.784,166.663,51.044,159.302
C09630=1021.013,-5.331,-100.769,166.660,51.049,159.302
C09631=1021.007,-5.612,-100.754,166.657,51.055,159.303
C09632=1021.001,-5.861,-100.741,166.654,51.060,159.303
C09633=1020.995,-6.111,-100.727,166.652,51.065,159.303
C09634=1020.989,-6.361,-100.713,166.648,51.070,159.304
C09635=1020.983,-6.610,-100.700,166.646,51.075,159.304
C09636=1020.978,-6.860,-100.687,166.643,51.080,159.305
C09637=1020.971,-7.110,-100.674,166.641,51.085,159.305
C09638=1020.966,-7.359,-100.660,166.637,51.089,159.305
C09639=1020.960,-7.608,-100.646,166.635,51.094,159.306
C09640=1020.954,-7.858,-100.633,166.632,51.099,159.306
C09641=1020.948,-8.108,-100.620,166.630,51.104,159.307
C09642=1020.943,-8.358,-100.606,166.626,51.109,159.307
C09643=1020.937,-8.607,-100.593,166.624,51.113,159.308
C09644=1020.930,-8.856,-100.580,166.622,51.118,159.308
C09645=1020.925,-9.106,-100.566,166.618,51.124,159.308
C09646=1020.919,-9.355,-100.553,166.616,51.128,159.309
C09647=1020.913,-9.605,-100.539,166.613,51.133,159.309
C09648=1020.907,-9.854,-100.526,166.610,51.138,159.310
C09649=1020.902,-10.105,-100.513,166.607,51.143,159.310
C09650=1020.896,-10.354,-100.500,166.605,51.148,159.311
C09651=1020.890,-10.603,-100.486,166.601,51.152,159.311
C09652=1020.885,-10.853,-100.473,166.599,51.157,159.311
C09653=1020.878,-11.103,-100.460,166.596,51.162,159.312
C09654=1020.873,-11.352,-100.446,166.593,51.167,159.312
C09655=1020.867,-11.602,-100.433,166.590,51.172,159.312
C09656=1020.861,-11.852,-100.420,166.588,51.177,159.313
C09657=1020.855,-12.101,-100.406,166.585,51.182,159.313
C09658=1020.850,-12.351,-100.393,166.582,51.186,159.314
C09659=1020.844,-12.600,-100.380,166.579,51.191,159.314
C09660=1020.838,-12.850,-100.366,166.577,51.196,159.315
C09661=1020.832,-13.100,-100.354,166.573,51.200,159.315
C09662=1020.826,-13.349,-100.340,166.571,51.205,159.315
C09663=1020.821,-13.599,-100.326,166.569,51.210,159.316
C09664=1020.815,-13.848,-100.314,166.565,51.215,159.316
C09665=1020.810,-14.097,-100.300,166.563,51.220,159.316
C09666=1020.804,-14.347,-100.288,166.560,51.224,159.317
C09667=1020.799,-14.597,-100.274,166.557,51.229,159.317
C09668=1020.792,-14.846,-100.261,166.554,51.234,159.318
C09669=1020.786,-15.096,-100.248,166.552,51.238,159.318
C09670=1020.781,-15.345,-100.234,166.548,51.244,159.318
C09671=1020.775,-15.595,-100.222,166.546,51.248,159.319
C09672=1020.770,-15.845,-100.208,166.544,51.253,159.319
C09673=1020.764,-16.095,-100.195,166.540,51.258,159.319
C09674=1020.757,-16.344,-100.182,166.537,51.263,159.320
C09675=1020.752,-16.593,-100.170,166.535,51.268,159.320
C09676=1020.746,-16.843,-100.157,166.531,51.272,159.321
C09677=1020.741,-17.093,-100.143,166.529,51.277,159.321
C09678=1020.735,-17.343,-100.131,166.526,51.282,159.321
C09679=1020.729,-17.592,-100.118,166.524,51.287,159.322
C09680=1020.723,-17.842,-100.105,166.520,51.292,159.322
C09681=1020.717,-18.092,-100.092,166.518,51.297,159.323
C09682=1020.711,-18.341,-100.079,166.515,51.302,159.323
C09683=1020.706,-18.590,-100.066,166.513,51.307,159.324
C09684=1020.700,-18.840,-100.053,166.509,51.311,159.324
C09685=1020.694,-19.090,-100.041,166.507,51.316,159.324
C09686=1020.688,-19.339,-100.028,166.504,51.321,159.325
C09687=1020.682,-19.589,-100.015,166.502,51.326,159.325
C09688=1020.676,-19.839,-100.002,166.498,51.331,159.325
C09689=1020.671,-20.088,-99.990,166.495,51.336,159.326
C09690=1020.665,-20.337,-99.976,166.493,51.341,159.326
C09691=1020.659,-20.587,-99.964,166.489,51.345,159.326
C09692=1020.653,-20.867,-99.949,166.486,51.351,159.327
C09693=1020.646,-21.146,-99.935,166.483,51.357,159.327
C09694=1020.640,-21.424,-99.921,166.480,51.362,159.328
C09695=1020.633,-21.704,-99.907,166.477,51.367,159.328
C09696=1020.627,-21.953,-99.894,166.475,51.372,159.329
C09697=1020.621,-22.203,-99.881,166.471,51.377,159.329
C09698=1020.617,-22.452,-99.868,166.469,51.381,159.329
C09699=1020.611,-22.702,-99.856,166.466,51.387,159.330
C09700=1020.604,-22.951,-99.842,166.463,51.391,159.330
C09701=1020.599,-23.201,-99.830,166.460,51.396,159.330
C09702=1020.593,-23.451,-99.817,166.458,51.401,159.331
C09703=1020.587,-23.700,-99.805,166.454,51.405,159.331
C09704=1020.581,-23.950,-99.793,166.452,51.410,159.332
C09705=1020.576,-24.200,-99.779,166.448,51.415,159.332
C09706=1020.571,-24.449,-99.767,166.446,51.420,159.332
C09707=1020.565,-24.699,-99.754,166.443,51.425,159.333
C09708=1020.559,-24.949,-99.741,166.441,51.429,159.333
C09709=1020.553,-25.199,-99.729,166.437,51.434,159.333
C09710=1020.547,-25.447,-99.716,166.435,51.438,159.334
C09711=1020.541,-25.697,-99.703,166.432,51.444,159.334
C09712=1020.536,-25.947,-99.690,166.429,51.449,159.335
C09713=1020.531,-26.197,-99.678,166.426,51.453,159.335
C09714=1020.525,-26.446,-99.666,166.424,51.458,159.335
C09715=1020.519,-26.696,-99.653,166.420,51.463,159.335
C09716=1020.513,-26.946,-99.640,166.418,51.467,159.336
C09717=1020.508,-27.195,-99.628,166.414,51.472,159.336
C09718=1020.502,-27.445,-99.615,166.412,51.477,159.337
C09719=1020.496,-27.695,-99.602,166.409,51.481,159.337
C09720=1020.490,-27.944,-99.590,166.407,51.486,159.337
C09721=1020.485,-28.194,-99.578,166.403,51.492,159.338
C09722=1020.479,-28.443,-99.565,166.401,51.496,159.338
C09723=1020.473,-28.693,-99.553,166.398,51.501,159.338
C09724=1020.467,-28.943,-99.540,166.394,51.506,159.339
C09725=1020.462,-29.193,-99.529,166.392,51.511,159.339
C09726=1020.456,-29.442,-99.517,166.389,51.516,159.339
C09727=1020.450,-29.692,-99.504,166.387,51.521,159.340
C09728=1020.444,-29.942,-99.492,166.383,51.526,159.340
C09729=1020.439,-30.191,-99.480,166.381,51.530,159.341
C09730=1020.433,-30.441,-99.467,166.378,51.535,159.341
C09731=1020.427,-30.691,-99.455,166.374,51.540,159.341
C09732=1020.421,-30.939,-99.443,166.372,51.545,159.342
C09733=1020.415,-31.189,-99.430,166.369,51.550,159.342
C09734=1020.409,-31.439,-99.418,166.367,51.555,159.343
C09735=1020.404,-31.688,-99.406,166.363,51.559,159.343
C09736=1020.398,-31.939,-99.394,166.361,51.564,159.343
C09737=1020.393,-32.188,-99.382,166.357,51.569,159.343
C09738=1020.387,-32.438,-99.369,166.355,51.574,159.344
C09739=1020.380,-32.688,-99.357,166.352,51.579,159.344
C09740=1020.375,-32.937,-99.345,166.348,51.583,159.344
C09741=1020.369,-33.187,-99.332,166.346,51.588,159.345
C09742=1020.364,-33.436,-99.320,166.343,51.593,159.345
C09743=1020.358,-33.686,-99.308,166.341,51.598,159.346
C09744=1020.353,-33.935,-99.296,166.337,51.603,159.346
C09745=1020.346,-34.185,-99.284,166.335,51.607,159.346
C09746=1020.340,-34.435,-99.272,166.332,51.613,159.347
C09747=1020.335,-34.684,-99.259,166.329,51.617,159.347
C09748=1020.329,-34.935,-99.248,166.326,51.622,159.347
C09749=1020.324,-35.184,-99.235,166.322,51.627,159.348
C09750=1020.318,-35.434,-99.223,166.320,51.631,159.348
C09751=1020.312,-35.683,-99.211,166.317,51.636,159.348
C09752=1020.306,-35.933,-99.199,166.314,51.641,159.349
C09753=1020.301,-36.182,-99.187,166.311,51.646,159.349
C09754=1020.295,-36.432,-99.175,166.309,51.650,159.349
C09755=1020.290,-36.681,-99.163,166.306,51.656,159.350
C09756=1020.283,-36.960,-99.149,166.302,51.661,159.350
C09757=1020.277,-37.238,-99.136,166.299,51.666,159.351
C09758=1020.271,-37.516,-99.123,166.296,51.671,159.351
C09759=1020.264,-37.794,-99.109,166.293,51.677,159.351
C09760=1020.258,-38.044,-99.097,166.290,51.681,159.352
C09761=1020.253,-38.294,-99.085,166.287,51.686,159.352
C09762=1020.247,-38.544,-99.073,166.285,51.690,159.352
C09763=1020.242,-38.793,-99.061,166.281,51.695,159.352
C09764=1020.236,-39.043,-99.049,166.279,51.700,159.353
C09765=1020.230,-39.292,-99.037,166.275,51.704,159.353
C09766=1020.225,-39.543,-99.025,166.272,51.710,159.354
C09767=1020.219,-39.792,-99.013,166.270,51.715,159.354
C09768=1020.214,-40.041,-99.002,166.267,51.719,159.354
C09769=1020.208,-40.291,-98.989,166.264,51.724,159.355
C09770=1020.202,-40.541,-98.979,166.261,51.729,159.355
C09771=1020.196,-40.791,-98.966,166.258,51.734,159.355
C09772=1020.190,-41.040,-98.955,166.256,51.739,159.356
C09773=1020.184,-41.290,-98.943,166.252,51.743,159.356
C09774=1020.179,-41.539,-98.932,166.250,51.748,159.356
C09775=1020.173,-41.789,-98.920,166.247,51.754,159.357
C09776=1020.168,-42.039,-98.908,166.243,51.758,159.357
C09777=1020.162,-42.288,-98.896,166.241,51.763,159.357
C09778=1020.156,-42.538,-98.884,166.237,51.768,159.358
C09779=1020.150,-42.788,-98.873,166.235,51.773,159.358
C09780=1020.145,-43.037,-98.861,166.232,51.777,159.358
C09781=1020.139,-43.287,-98.850,166.229,51.782,159.359
C09782=1020.133,-43.537,-98.838,166.226,51.787,159.359
C09783=1020.127,-43.787,-98.827,166.223,51.792,159.359
C09784=1020.122,-44.036,-98.814,166.221,51.797,159.360
C09785=1020.116,-44.285,-98.803,166.217,51.801,159.360
C09786=1020.110,-44.536,-98.792,166.214,51.807,159.360
C09787=1020.105,-44.785,-98.779,166.212,51.811,159.361
C09788=1020.099,-45.035,-98.769,166.208,51.816,159.361
C09789=1020.094,-45.285,-98.757,166.206,51.820,159.361
C09790=1020.088,-45.534,-98.745,166.203,51.826,159.362
C09791=1020.083,-45.784,-98.734,166.200,51.830,159.362
C09792=1020.076,-46.033,-98.722,166.197,51.835,159.362
C09793=1020.071,-46.283,-98.710,166.193,51.840,159.363
C09794=1020.065,-46.533,-98.699,166.191,51.845,159.363
C09795=1020.059,-46.782,-98.687,166.188,51.849,159.363
C09796=1020.054,-47.032,-98.676,166.186,51.854,159.364
C09797=1020.049,-47.282,-98.664,166.182,51.859,159.364
C09798=1020.042,-47.532,-98.653,166.180,51.863,159.364
C09799=1020.037,-47.781,-98.641,166.176,51.868,159.365
C09800=1020.031,-48.031,-98.630,166.173,51.873,159.365
C09801=1020.026,-48.280,-98.619,166.171,51.878,159.365
C09802=1020.020,-48.530,-98.606,166.167,51.882,159.365
C09803=1020.015,-48.780,-98.595,166.165,51.887,159.366
C09804=1020.010,-49.030,-98.584,166.161,51.892,159.366
C09805=1020.004,-49.279,-98.573,166.159,51.896,159.366
C09806=1019.998,-49.529,-98.560,166.156,51.901,159.367
C09807=1019.992,-49.778,-98.549,166.153,51.906,159.367
C09808=1019.987,-50.028,-98.538,166.150,51.911,159.367
C09809=1019.982,-50.278,-98.527,166.147,51.915,159.367
C09810=1019.976,-50.528,-98.515,166.144,51.920,159.368
C09811=1019.970,-50.777,-98.504,166.141,51.925,159.368
C09812=1019.965,-51.027,-98.492,166.138,51.929,159.368
C09813=1019.959,-51.276,-98.481,166.135,51.934,159.369
C09814=1019.953,-51.527,-98.470,166.132,51.940,159.369
C09815=1019.947,-51.776,-98.459,166.130,51.944,159.369
C09816=1019.941,-52.026,-98.448,166.126,51.949,159.370
C09817=1019.936,-52.275,-98.437,166.123,51.955,159.370
C09818=1019.930,-52.525,-98.427,166.121,51.959,159.370
C09819=1019.924,-52.775,-98.415,166.118,51.964,159.371
C09820=1019.918,-53.053,-98.403,166.114,51.969,159.371
C09821=1019.912,-53.332,-98.390,166.111,51.975,159.372
C09822=1019.905,-53.610,-98.378,166.107,51.980,159.372
C09823=1019.899,-53.889,-98.366,166.104,51.986,159.372
C09824=1019.893,-54.138,-98.355,166.101,51.991,159.373
C09825=1019.887,-54.388,-98.344,166.099,51.996,159.373
C09826=1019.881,-54.638,-98.333,166.095,52.001,159.373
C09827=1019.876,-54.888,-98.323,166.092,52.006,159.374
C09828=1019.870,-55.138,-98.312,166.090,52.010,159.374
C09829=1019.864,-55.387,-98.301,166.086,52.015,159.374
C09830=1019.858,-55.637,-98.290,166.083,52.021,159.375
C09831=1019.853,-55.886,-98.278,166.081,52.025,159.375
C09832=1019.848,-56.136,-98.268,166.078,52.030,159.375
C09833=1019.841,-56.386,-98.256,166.074,52.035,159.375
///RCONF 1,0,0,1,0,0,0,0,0,0,0,0,0,0,0,0,0,0,0,0,0,0,0,0
C09834=1019.836,-56.636,-98.245,166.072,52.040,159.376
C09835=1019.830,-56.885,-98.235,166.068,52.044,159.376
C09836=1019.824,-57.135,-98.224,166.065,52.050,159.376
C09837=1019.819,-57.385,-98.214,166.063,52.054,159.377
C09838=1019.813,-57.634,-98.203,166.060,52.059,159.377
C09839=1019.807,-57.884,-98.192,166.056,52.064,159.377
C09840=1019.802,-58.133,-98.180,166.054,52.069,159.378
C09841=1019.797,-58.384,-98.170,166.050,52.073,159.378
C09842=1019.791,-58.633,-98.159,166.048,52.078,159.378
C09843=1019.785,-58.883,-98.148,166.045,52.083,159.378
C09844=1019.779,-59.133,-98.137,166.042,52.088,159.379
C09845=1019.773,-59.382,-98.126,166.039,52.092,159.379
C09846=1019.768,-59.632,-98.116,166.036,52.098,159.379
C09847=1019.762,-59.882,-98.105,166.032,52.102,159.380
C09848=1019.756,-60.131,-98.094,166.030,52.107,159.380
C09849=1019.750,-60.381,-98.083,166.027,52.112,159.380
C09850=1019.746,-60.631,-98.073,166.024,52.117,159.381
C09851=1019.740,-60.881,-98.062,166.021,52.122,159.381
C09852=1019.734,-61.130,-98.051,166.018,52.127,159.381
C09853=1019.729,-61.380,-98.040,166.016,52.131,159.382
C09854=1019.723,-61.630,-98.030,166.012,52.136,159.382
C09855=1019.717,-61.879,-98.019,166.009,52.141,159.382
C09856=1019.712,-62.129,-98.008,166.006,52.145,159.382
C09857=1019.706,-62.379,-97.998,166.003,52.151,159.383
C09858=1019.700,-62.628,-97.987,166.000,52.155,159.383
C09859=1019.695,-62.878,-97.976,165.998,52.160,159.383
C09860=1019.689,-63.128,-97.966,165.994,52.165,159.384
C09861=1019.684,-63.378,-97.955,165.992,52.169,159.384
C09862=1019.679,-63.627,-97.944,165.988,52.174,159.384
C09863=1019.673,-63.877,-97.934,165.985,52.179,159.384
C09864=1019.667,-64.127,-97.923,165.982,52.183,159.385
C09865=1019.662,-64.376,-97.912,165.979,52.189,159.385
C09866=1019.656,-64.627,-97.902,165.977,52.193,159.385
C09867=1019.650,-64.876,-97.891,165.974,52.198,159.386
C09868=1019.646,-65.125,-97.881,165.970,52.203,159.386
C09869=1019.640,-65.375,-97.870,165.968,52.207,159.386
C09870=1019.634,-65.624,-97.859,165.964,52.212,159.386
C09871=1019.629,-65.874,-97.849,165.962,52.217,159.387
C09872=1019.623,-66.124,-97.838,165.958,52.221,159.387
C09873=1019.618,-66.374,-97.828,165.955,52.226,159.387
C09874=1019.612,-66.624,-97.817,165.953,52.231,159.387
C09875=1019.607,-66.873,-97.806,165.949,52.235,159.388
C09876=1019.601,-67.123,-97.796,165.947,52.240,159.388
C09877=1019.596,-67.373,-97.785,165.944,52.245,159.388
C09878=1019.591,-67.622,-97.775,165.941,52.249,159.389
C09879=1019.585,-67.872,-97.764,165.938,52.254,159.389
C09880=1019.580,-68.122,-97.754,165.934,52.259,159.389
C09881=1019.574,-68.371,-97.743,165.932,52.263,159.389
C09882=1019.568,-68.622,-97.733,165.928,52.268,159.389
C09883=1019.563,-68.871,-97.722,165.926,52.272,159.390
C09884=1019.557,-69.151,-97.711,165.923,52.278,159.390
C09885=1019.551,-69.431,-97.699,165.919,52.283,159.390
C09886=1019.544,-69.710,-97.687,165.915,52.289,159.391
C09887=1019.538,-69.990,-97.675,165.912,52.294,159.391
C09888=1019.533,-70.240,-97.665,165.910,52.298,159.391
C09889=1019.528,-70.489,-97.654,165.906,52.303,159.391
C09890=1019.522,-70.739,-97.644,165.904,52.307,159.392
C09891=1019.517,-70.989,-97.634,165.900,52.312,159.392
C09892=1019.512,-71.239,-97.623,165.897,52.317,159.392
C09893=1019.506,-71.489,-97.613,165.895,52.321,159.393
C09894=1019.501,-71.738,-97.602,165.891,52.326,159.393
C09895=1019.496,-71.988,-97.592,165.889,52.330,159.393
C09896=1019.490,-72.238,-97.582,165.885,52.335,159.393
C09897=1019.485,-72.487,-97.571,165.883,52.340,159.394
C09898=1019.480,-72.737,-97.561,165.879,52.345,159.394
C09899=1019.474,-72.987,-97.551,165.877,52.349,159.394
C09900=1019.469,-73.236,-97.540,165.873,52.353,159.394
C09901=1019.463,-73.486,-97.530,165.871,52.358,159.394
C09902=1019.458,-73.735,-97.519,165.867,52.362,159.395
C09903=1019.453,-73.985,-97.509,165.865,52.367,159.395
C09904=1019.447,-74.235,-97.499,165.862,52.372,159.395
C09905=1019.442,-74.486,-97.489,165.858,52.377,159.395
C09906=1019.437,-74.734,-97.478,165.856,52.381,159.396
C09907=1019.431,-74.984,-97.468,165.853,52.386,159.396
C09908=1019.425,-75.234,-97.459,165.850,52.390,159.396
C09909=1019.420,-75.484,-97.448,165.847,52.395,159.396
C09910=1019.415,-75.734,-97.439,165.844,52.400,159.397
C09911=1019.409,-75.984,-97.428,165.841,52.405,159.397
C09912=1019.403,-76.233,-97.418,165.837,52.409,159.397
C09913=1019.398,-76.482,-97.408,165.834,52.415,159.397
C09914=1019.393,-76.733,-97.398,165.832,52.419,159.398
C09915=1019.387,-76.983,-97.388,165.828,52.424,159.398
C09916=1019.382,-77.232,-97.379,165.826,52.429,159.398
C09917=1019.376,-77.482,-97.369,165.823,52.433,159.399
C09918=1019.371,-77.732,-97.359,165.819,52.438,159.399
C09919=1019.365,-77.981,-97.349,165.817,52.442,159.399
C09920=1019.360,-78.231,-97.339,165.814,52.448,159.399
C09921=1019.354,-78.481,-97.329,165.810,52.452,159.399
C09922=1019.350,-78.731,-97.319,165.808,52.456,159.400
C09923=1019.343,-78.980,-97.309,165.805,52.462,159.400
C09924=1019.338,-79.230,-97.299,165.802,52.466,159.400
C09925=1019.333,-79.479,-97.289,165.798,52.471,159.400
C09926=1019.327,-79.729,-97.279,165.795,52.475,159.401
C09927=1019.321,-79.979,-97.269,165.793,52.480,159.401
C09928=1019.316,-80.229,-97.259,165.789,52.485,159.401
C09929=1019.311,-80.479,-97.250,165.787,52.489,159.402
C09930=1019.306,-80.729,-97.241,165.784,52.495,159.402
C09931=1019.300,-80.979,-97.231,165.780,52.499,159.402
C09932=1019.294,-81.228,-97.221,165.777,52.504,159.402
C09933=1019.288,-81.478,-97.212,165.775,52.509,159.403
C09934=1019.283,-81.728,-97.202,165.771,52.514,159.403
C09935=1019.277,-81.977,-97.193,165.768,52.519,159.403
C09936=1019.272,-82.227,-97.182,165.766,52.523,159.403
C09937=1019.266,-82.477,-97.173,165.762,52.529,159.404
C09938=1019.261,-82.727,-97.164,165.759,52.533,159.404
C09939=1019.255,-82.976,-97.154,165.756,52.538,159.404
C09940=1019.250,-83.226,-97.144,165.753,52.543,159.404
C09941=1019.244,-83.476,-97.135,165.750,52.548,159.405
C09942=1019.240,-83.726,-97.126,165.747,52.552,159.405
C09943=1019.233,-83.975,-97.116,165.744,52.557,159.405
C09944=1019.229,-84.225,-97.106,165.741,52.562,159.405
C09945=1019.222,-84.475,-97.097,165.739,52.567,159.406
C09946=1019.217,-84.724,-97.088,165.735,52.572,159.406
C09947=1019.212,-84.975,-97.078,165.732,52.576,159.406
C09948=1019.206,-85.256,-97.067,165.729,52.582,159.406
C09949=1019.199,-85.537,-97.057,165.725,52.587,159.407
C09950=1019.193,-85.820,-97.047,165.721,52.593,159.407
C09951=1019.187,-86.101,-97.036,165.718,52.598,159.407
C09952=1019.181,-86.351,-97.026,165.716,52.602,159.408
C09953=1019.176,-86.600,-97.016,165.712,52.607,159.408
C09954=1019.171,-86.851,-97.007,165.709,52.612,159.408
C09955=1019.166,-87.100,-96.998,165.707,52.617,159.408
C09956=1019.160,-87.350,-96.988,165.703,52.621,159.408
C09957=1019.155,-87.600,-96.979,165.700,52.627,159.409
C09958=1019.149,-87.850,-96.969,165.698,52.631,159.409
C09959=1019.143,-88.099,-96.960,165.694,52.636,159.409
C09960=1019.139,-88.349,-96.951,165.691,52.641,159.410
C09961=1019.133,-88.599,-96.942,165.688,52.645,159.410
C09962=1019.128,-88.848,-96.932,165.685,52.650,159.410
C09963=1019.122,-89.098,-96.923,165.681,52.655,159.410
C09964=1019.117,-89.348,-96.913,165.679,52.660,159.411
C09965=1019.111,-89.598,-96.904,165.676,52.664,159.411
C09966=1019.106,-89.847,-96.895,165.672,52.669,159.411
C09967=1019.101,-90.097,-96.885,165.670,52.674,159.411
C09968=1019.095,-90.347,-96.876,165.667,52.679,159.411
C09969=1019.090,-90.597,-96.867,165.664,52.683,159.412
C09970=1019.084,-90.847,-96.858,165.661,52.688,159.412
C09971=1019.079,-91.096,-96.848,165.658,52.693,159.412
C09972=1019.074,-91.346,-96.839,165.655,52.697,159.412
C09973=1019.068,-91.596,-96.830,165.652,52.702,159.413
C09974=1019.063,-91.845,-96.820,165.648,52.707,159.413
C09975=1019.058,-92.095,-96.812,165.646,52.712,159.413
C09976=1019.052,-92.345,-96.801,165.643,52.716,159.413
C09977=1019.047,-92.595,-96.793,165.640,52.721,159.414
C09978=1019.042,-92.844,-96.783,165.637,52.725,159.414
C09979=1019.036,-93.095,-96.774,165.633,52.730,159.414
C09980=1019.031,-93.344,-96.765,165.631,52.735,159.414
C09981=1019.026,-93.594,-96.756,165.628,52.740,159.414
C09982=1019.020,-93.844,-96.746,165.624,52.744,159.415
C09983=1019.016,-94.094,-96.737,165.622,52.749,159.415
C09984=1019.010,-94.343,-96.729,165.618,52.753,159.415
C09985=1019.004,-94.593,-96.719,165.616,52.758,159.415
C09986=1019.000,-94.843,-96.710,165.612,52.763,159.416
C09987=1018.994,-95.092,-96.701,165.609,52.768,159.416
C09988=1018.990,-95.342,-96.692,165.606,52.772,159.416
C09989=1018.983,-95.592,-96.682,165.603,52.777,159.416
C09990=1018.978,-95.842,-96.674,165.601,52.781,159.416
C09991=1018.974,-96.092,-96.665,165.597,52.786,159.417
C09992=1018.968,-96.341,-96.656,165.595,52.791,159.417
C09993=1018.963,-96.592,-96.646,165.591,52.795,159.417
C09994=1018.957,-96.841,-96.637,165.588,52.800,159.417
C09995=1018.952,-97.091,-96.629,165.585,52.804,159.417
C09996=1018.948,-97.341,-96.619,165.582,52.809,159.418
//INST
///DATE 2021/06/17 10:59
///ATTR SC,RW,RJ
////FRAME ROBOT
///GROUP1 RB1
NOP
MOVL C00000 V=800.0 PL=0
MOVL C00001 V=800.0 PL=0
MOVL C00002 V=800.0 PL=0
MOVL C00003 V=800.0 PL=0
MOVL C00004 V=800.0 PL=0
MOVL C00005 V=800.0 PL=0
MOVL C00006 V=800.0 PL=0
MOVL C00007 V=800.0 PL=0
MOVL C00008 V=800.0 PL=0
MOVL C00009 V=800.0 PL=0
MOVL C00010 V=800.0 PL=0
MOVL C00011 V=800.0 PL=0
MOVL C00012 V=800.0 PL=0
MOVL C00013 V=800.0 PL=0
MOVL C00014 V=800.0 PL=0
MOVL C00015 V=800.0 PL=0
MOVL C00016 V=800.0 PL=0
MOVL C00017 V=800.0 PL=0
MOVL C00018 V=800.0 PL=0
MOVL C00019 V=800.0 PL=0
MOVL C00020 V=800.0 PL=0
MOVL C00021 V=800.0 PL=0
MOVL C00022 V=800.0 PL=0
MOVL C00023 V=800.0 PL=0
MOVL C00024 V=800.0 PL=0
MOVL C00025 V=800.0 PL=0
MOVL C00026 V=800.0 PL=0
MOVL C00027 V=800.0 PL=0
MOVL C00028 V=800.0 PL=0
MOVL C00029 V=800.0 PL=0
MOVL C00030 V=800.0 PL=0
MOVL C00031 V=800.0 PL=0
MOVL C00032 V=800.0 PL=0
MOVL C00033 V=800.0 PL=0
MOVL C00034 V=800.0 PL=0
MOVL C00035 V=800.0 PL=0
MOVL C00036 V=800.0 PL=0
MOVL C00037 V=800.0 PL=0
MOVL C00038 V=800.0 PL=0
MOVL C00039 V=800.0 PL=0
MOVL C00040 V=800.0 PL=0
MOVL C00041 V=800.0 PL=0
MOVL C00042 V=800.0 PL=0
MOVL C00043 V=800.0 PL=0
MOVL C00044 V=800.0 PL=0
MOVL C00045 V=800.0 PL=0
MOVL C00046 V=800.0 PL=0
MOVL C00047 V=800.0 PL=0
MOVL C00048 V=800.0 PL=0
MOVL C00049 V=800.0 PL=0
MOVL C00050 V=800.0 PL=0
MOVL C00051 V=800.0 PL=0
MOVL C00052 V=800.0 PL=0
MOVL C00053 V=800.0 PL=0
MOVL C00054 V=800.0 PL=0
MOVL C00055 V=800.0 PL=0
MOVL C00056 V=800.0 PL=0
MOVL C00057 V=800.0 PL=0
MOVL C00058 V=800.0 PL=0
MOVL C00059 V=800.0 PL=0
MOVL C00060 V=800.0 PL=0
MOVL C00061 V=800.0 PL=0
MOVL C00062 V=800.0 PL=0
MOVL C00063 V=800.0 PL=0
MOVL C00064 V=800.0 PL=0
MOVL C00065 V=800.0 PL=0
MOVL C00066 V=800.0 PL=0
MOVL C00067 V=800.0 PL=0
MOVL C00068 V=800.0 PL=0
MOVL C00069 V=800.0 PL=0
MOVL C00070 V=800.0 PL=0
MOVL C00071 V=800.0 PL=0
MOVL C00072 V=800.0 PL=0
MOVL C00073 V=800.0 PL=0
MOVL C00074 V=800.0 PL=0
MOVL C00075 V=800.0 PL=0
MOVL C00076 V=800.0 PL=0
MOVL C00077 V=800.0 PL=0
MOVL C00078 V=800.0 PL=0
MOVL C00079 V=800.0 PL=0
MOVL C00080 V=800.0 PL=0
MOVL C00081 V=800.0 PL=0
MOVL C00082 V=800.0 PL=0
MOVL C00083 V=800.0 PL=0
MOVL C00084 V=800.0 PL=0
MOVL C00085 V=800.0 PL=0
MOVL C00086 V=800.0 PL=0
MOVL C00087 V=800.0 PL=0
MOVL C00088 V=800.0 PL=0
MOVL C00089 V=800.0 PL=0
MOVL C00090 V=800.0 PL=0
MOVL C00091 V=800.0 PL=0
MOVL C00092 V=800.0 PL=0
MOVL C00093 V=800.0 PL=0
MOVL C00094 V=800.0 PL=0
MOVL C00095 V=800.0 PL=0
MOVL C00096 V=800.0 PL=0
MOVL C00097 V=800.0 PL=0
MOVL C00098 V=800.0 PL=0
MOVL C00099 V=800.0 PL=0
MOVL C00100 V=800.0 PL=0
MOVL C00101 V=800.0 PL=0
MOVL C00102 V=800.0 PL=0
MOVL C00103 V=800.0 PL=0
MOVL C00104 V=800.0 PL=0
MOVL C00105 V=800.0 PL=0
MOVL C00106 V=800.0 PL=0
MOVL C00107 V=800.0 PL=0
MOVL C00108 V=800.0 PL=0
MOVL C00109 V=800.0 PL=0
MOVL C00110 V=800.0 PL=0
MOVL C00111 V=800.0 PL=0
MOVL C00112 V=800.0 PL=0
MOVL C00113 V=800.0 PL=0
MOVL C00114 V=800.0 PL=0
MOVL C00115 V=800.0 PL=0
MOVL C00116 V=800.0 PL=0
MOVL C00117 V=800.0 PL=0
MOVL C00118 V=800.0 PL=0
MOVL C00119 V=800.0 PL=0
MOVL C00120 V=800.0 PL=0
MOVL C00121 V=800.0 PL=0
MOVL C00122 V=800.0 PL=0
MOVL C00123 V=800.0 PL=0
MOVL C00124 V=800.0 PL=0
MOVL C00125 V=800.0 PL=0
MOVL C00126 V=800.0 PL=0
MOVL C00127 V=800.0 PL=0
MOVL C00128 V=800.0 PL=0
MOVL C00129 V=800.0 PL=0
MOVL C00130 V=800.0 PL=0
MOVL C00131 V=800.0 PL=0
MOVL C00132 V=800.0 PL=0
MOVL C00133 V=800.0 PL=0
MOVL C00134 V=800.0 PL=0
MOVL C00135 V=800.0 PL=0
MOVL C00136 V=800.0 PL=0
MOVL C00137 V=800.0 PL=0
MOVL C00138 V=800.0 PL=0
MOVL C00139 V=800.0 PL=0
MOVL C00140 V=800.0 PL=0
MOVL C00141 V=800.0 PL=0
MOVL C00142 V=800.0 PL=0
MOVL C00143 V=800.0 PL=0
MOVL C00144 V=800.0 PL=0
MOVL C00145 V=800.0 PL=0
MOVL C00146 V=800.0 PL=0
MOVL C00147 V=800.0 PL=0
MOVL C00148 V=800.0 PL=0
MOVL C00149 V=800.0 PL=0
MOVL C00150 V=800.0 PL=0
MOVL C00151 V=800.0 PL=0
MOVL C00152 V=800.0 PL=0
MOVL C00153 V=800.0 PL=0
MOVL C00154 V=800.0 PL=0
MOVL C00155 V=800.0 PL=0
MOVL C00156 V=800.0 PL=0
MOVL C00157 V=800.0 PL=0
MOVL C00158 V=800.0 PL=0
MOVL C00159 V=800.0 PL=0
MOVL C00160 V=800.0 PL=0
MOVL C00161 V=800.0 PL=0
MOVL C00162 V=800.0 PL=0
MOVL C00163 V=800.0 PL=0
MOVL C00164 V=800.0 PL=0
MOVL C00165 V=800.0 PL=0
MOVL C00166 V=800.0 PL=0
MOVL C00167 V=800.0 PL=0
MOVL C00168 V=800.0 PL=0
MOVL C00169 V=800.0 PL=0
MOVL C00170 V=800.0 PL=0
MOVL C00171 V=800.0 PL=0
MOVL C00172 V=800.0 PL=0
MOVL C00173 V=800.0 PL=0
MOVL C00174 V=800.0 PL=0
MOVL C00175 V=800.0 PL=0
MOVL C00176 V=800.0 PL=0
MOVL C00177 V=800.0 PL=0
MOVL C00178 V=800.0 PL=0
MOVL C00179 V=800.0 PL=0
MOVL C00180 V=800.0 PL=0
MOVL C00181 V=800.0 PL=0
MOVL C00182 V=800.0 PL=0
MOVL C00183 V=800.0 PL=0
MOVL C00184 V=800.0 PL=0
MOVL C00185 V=800.0 PL=0
MOVL C00186 V=800.0 PL=0
MOVL C00187 V=800.0 PL=0
MOVL C00188 V=800.0 PL=0
MOVL C00189 V=800.0 PL=0
MOVL C00190 V=800.0 PL=0
MOVL C00191 V=800.0 PL=0
MOVL C00192 V=800.0 PL=0
MOVL C00193 V=800.0 PL=0
MOVL C00194 V=800.0 PL=0
MOVL C00195 V=800.0 PL=0
MOVL C00196 V=800.0 PL=0
MOVL C00197 V=800.0 PL=0
MOVL C00198 V=800.0 PL=0
MOVL C00199 V=800.0 PL=0
MOVL C00200 V=800.0 PL=0
MOVL C00201 V=800.0 PL=0
MOVL C00202 V=800.0 PL=0
MOVL C00203 V=800.0 PL=0
MOVL C00204 V=800.0 PL=0
MOVL C00205 V=800.0 PL=0
MOVL C00206 V=800.0 PL=0
MOVL C00207 V=800.0 PL=0
MOVL C00208 V=800.0 PL=0
MOVL C00209 V=800.0 PL=0
MOVL C00210 V=800.0 PL=0
MOVL C00211 V=800.0 PL=0
MOVL C00212 V=800.0 PL=0
MOVL C00213 V=800.0 PL=0
MOVL C00214 V=800.0 PL=0
MOVL C00215 V=800.0 PL=0
MOVL C00216 V=800.0 PL=0
MOVL C00217 V=800.0 PL=0
MOVL C00218 V=800.0 PL=0
MOVL C00219 V=800.0 PL=0
MOVL C00220 V=800.0 PL=0
MOVL C00221 V=800.0 PL=0
MOVL C00222 V=800.0 PL=0
MOVL C00223 V=800.0 PL=0
MOVL C00224 V=800.0 PL=0
MOVL C00225 V=800.0 PL=0
MOVL C00226 V=800.0 PL=0
MOVL C00227 V=800.0 PL=0
MOVL C00228 V=800.0 PL=0
MOVL C00229 V=800.0 PL=0
MOVL C00230 V=800.0 PL=0
MOVL C00231 V=800.0 PL=0
MOVL C00232 V=800.0 PL=0
MOVL C00233 V=800.0 PL=0
MOVL C00234 V=800.0 PL=0
MOVL C00235 V=800.0 PL=0
MOVL C00236 V=800.0 PL=0
MOVL C00237 V=800.0 PL=0
MOVL C00238 V=800.0 PL=0
MOVL C00239 V=800.0 PL=0
MOVL C00240 V=800.0 PL=0
MOVL C00241 V=800.0 PL=0
MOVL C00242 V=800.0 PL=0
MOVL C00243 V=800.0 PL=0
MOVL C00244 V=800.0 PL=0
MOVL C00245 V=800.0 PL=0
MOVL C00246 V=800.0 PL=0
MOVL C00247 V=800.0 PL=0
MOVL C00248 V=800.0 PL=0
MOVL C00249 V=800.0 PL=0
MOVL C00250 V=800.0 PL=0
MOVL C00251 V=800.0 PL=0
MOVL C00252 V=800.0 PL=0
MOVL C00253 V=800.0 PL=0
MOVL C00254 V=800.0 PL=0
MOVL C00255 V=800.0 PL=0
MOVL C00256 V=800.0 PL=0
MOVL C00257 V=800.0 PL=0
MOVL C00258 V=800.0 PL=0
MOVL C00259 V=800.0 PL=0
MOVL C00260 V=800.0 PL=0
MOVL C00261 V=800.0 PL=0
MOVL C00262 V=800.0 PL=0
MOVL C00263 V=800.0 PL=0
MOVL C00264 V=800.0 PL=0
MOVL C00265 V=800.0 PL=0
MOVL C00266 V=800.0 PL=0
MOVL C00267 V=800.0 PL=0
MOVL C00268 V=800.0 PL=0
MOVL C00269 V=800.0 PL=0
MOVL C00270 V=800.0 PL=0
MOVL C00271 V=800.0 PL=0
MOVL C00272 V=800.0 PL=0
MOVL C00273 V=800.0 PL=0
MOVL C00274 V=800.0 PL=0
MOVL C00275 V=800.0 PL=0
MOVL C00276 V=800.0 PL=0
MOVL C00277 V=800.0 PL=0
MOVL C00278 V=800.0 PL=0
MOVL C00279 V=800.0 PL=0
MOVL C00280 V=800.0 PL=0
MOVL C00281 V=800.0 PL=0
MOVL C00282 V=800.0 PL=0
MOVL C00283 V=800.0 PL=0
MOVL C00284 V=800.0 PL=0
MOVL C00285 V=800.0 PL=0
MOVL C00286 V=800.0 PL=0
MOVL C00287 V=800.0 PL=0
MOVL C00288 V=800.0 PL=0
MOVL C00289 V=800.0 PL=0
MOVL C00290 V=800.0 PL=0
MOVL C00291 V=800.0 PL=0
MOVL C00292 V=800.0 PL=0
MOVL C00293 V=800.0 PL=0
MOVL C00294 V=800.0 PL=0
MOVL C00295 V=800.0 PL=0
MOVL C00296 V=800.0 PL=0
MOVL C00297 V=800.0 PL=0
MOVL C00298 V=800.0 PL=0
MOVL C00299 V=800.0 PL=0
MOVL C00300 V=800.0 PL=0
MOVL C00301 V=800.0 PL=0
MOVL C00302 V=800.0 PL=0
MOVL C00303 V=800.0 PL=0
MOVL C00304 V=800.0 PL=0
MOVL C00305 V=800.0 PL=0
MOVL C00306 V=800.0 PL=0
MOVL C00307 V=800.0 PL=0
MOVL C00308 V=800.0 PL=0
MOVL C00309 V=800.0 PL=0
MOVL C00310 V=800.0 PL=0
MOVL C00311 V=800.0 PL=0
MOVL C00312 V=800.0 PL=0
MOVL C00313 V=800.0 PL=0
MOVL C00314 V=800.0 PL=0
MOVL C00315 V=800.0 PL=0
MOVL C00316 V=800.0 PL=0
MOVL C00317 V=800.0 PL=0
MOVL C00318 V=800.0 PL=0
MOVL C00319 V=800.0 PL=0
MOVL C00320 V=800.0 PL=0
MOVL C00321 V=800.0 PL=0
MOVL C00322 V=800.0 PL=0
MOVL C00323 V=800.0 PL=0
MOVL C00324 V=800.0 PL=0
MOVL C00325 V=800.0 PL=0
MOVL C00326 V=800.0 PL=0
MOVL C00327 V=800.0 PL=0
MOVL C00328 V=800.0 PL=0
MOVL C00329 V=800.0 PL=0
MOVL C00330 V=800.0 PL=0
MOVL C00331 V=800.0 PL=0
MOVL C00332 V=800.0 PL=0
MOVL C00333 V=800.0 PL=0
MOVL C00334 V=800.0 PL=0
MOVL C00335 V=800.0 PL=0
MOVL C00336 V=800.0 PL=0
MOVL C00337 V=800.0 PL=0
MOVL C00338 V=800.0 PL=0
MOVL C00339 V=800.0 PL=0
MOVL C00340 V=800.0 PL=0
MOVL C00341 V=800.0 PL=0
MOVL C00342 V=800.0 PL=0
MOVL C00343 V=800.0 PL=0
MOVL C00344 V=800.0 PL=0
MOVL C00345 V=800.0 PL=0
MOVL C00346 V=800.0 PL=0
MOVL C00347 V=800.0 PL=0
MOVL C00348 V=800.0 PL=0
MOVL C00349 V=800.0 PL=0
MOVL C00350 V=800.0 PL=0
MOVL C00351 V=800.0 PL=0
MOVL C00352 V=800.0 PL=0
MOVL C00353 V=800.0 PL=0
MOVL C00354 V=800.0 PL=0
MOVL C00355 V=800.0 PL=0
MOVL C00356 V=800.0 PL=0
MOVL C00357 V=800.0 PL=0
MOVL C00358 V=800.0 PL=0
MOVL C00359 V=800.0 PL=0
MOVL C00360 V=800.0 PL=0
MOVL C00361 V=800.0 PL=0
MOVL C00362 V=800.0 PL=0
MOVL C00363 V=800.0 PL=0
MOVL C00364 V=800.0 PL=0
MOVL C00365 V=800.0 PL=0
MOVL C00366 V=800.0 PL=0
MOVL C00367 V=800.0 PL=0
MOVL C00368 V=800.0 PL=0
MOVL C00369 V=800.0 PL=0
MOVL C00370 V=800.0 PL=0
MOVL C00371 V=800.0 PL=0
MOVL C00372 V=800.0 PL=0
MOVL C00373 V=800.0 PL=0
MOVL C00374 V=800.0 PL=0
MOVL C00375 V=800.0 PL=0
MOVL C00376 V=800.0 PL=0
MOVL C00377 V=800.0 PL=0
MOVL C00378 V=800.0 PL=0
MOVL C00379 V=800.0 PL=0
MOVL C00380 V=800.0 PL=0
MOVL C00381 V=800.0 PL=0
MOVL C00382 V=800.0 PL=0
MOVL C00383 V=800.0 PL=0
MOVL C00384 V=800.0 PL=0
MOVL C00385 V=800.0 PL=0
MOVL C00386 V=800.0 PL=0
MOVL C00387 V=800.0 PL=0
MOVL C00388 V=800.0 PL=0
MOVL C00389 V=800.0 PL=0
MOVL C00390 V=800.0 PL=0
MOVL C00391 V=800.0 PL=0
MOVL C00392 V=800.0 PL=0
MOVL C00393 V=800.0 PL=0
MOVL C00394 V=800.0 PL=0
MOVL C00395 V=800.0 PL=0
MOVL C00396 V=800.0 PL=0
MOVL C00397 V=800.0 PL=0
MOVL C00398 V=800.0 PL=0
MOVL C00399 V=800.0 PL=0
MOVL C00400 V=800.0 PL=0
MOVL C00401 V=800.0 PL=0
MOVL C00402 V=800.0 PL=0
MOVL C00403 V=800.0 PL=0
MOVL C00404 V=800.0 PL=0
MOVL C00405 V=800.0 PL=0
MOVL C00406 V=800.0 PL=0
MOVL C00407 V=800.0 PL=0
MOVL C00408 V=800.0 PL=0
MOVL C00409 V=800.0 PL=0
MOVL C00410 V=800.0 PL=0
MOVL C00411 V=800.0 PL=0
MOVL C00412 V=800.0 PL=0
MOVL C00413 V=800.0 PL=0
MOVL C00414 V=800.0 PL=0
MOVL C00415 V=800.0 PL=0
MOVL C00416 V=800.0 PL=0
MOVL C00417 V=800.0 PL=0
MOVL C00418 V=800.0 PL=0
MOVL C00419 V=800.0 PL=0
MOVL C00420 V=800.0 PL=0
MOVL C00421 V=800.0 PL=0
MOVL C00422 V=800.0 PL=0
MOVL C00423 V=800.0 PL=0
MOVL C00424 V=800.0 PL=0
MOVL C00425 V=800.0 PL=0
MOVL C00426 V=800.0 PL=0
MOVL C00427 V=800.0 PL=0
MOVL C00428 V=800.0 PL=0
MOVL C00429 V=800.0 PL=0
MOVL C00430 V=800.0 PL=0
MOVL C00431 V=800.0 PL=0
MOVL C00432 V=800.0 PL=0
MOVL C00433 V=800.0 PL=0
MOVL C00434 V=800.0 PL=0
MOVL C00435 V=800.0 PL=0
MOVL C00436 V=800.0 PL=0
MOVL C00437 V=800.0 PL=0
MOVL C00438 V=800.0 PL=0
MOVL C00439 V=800.0 PL=0
MOVL C00440 V=800.0 PL=0
MOVL C00441 V=800.0 PL=0
MOVL C00442 V=800.0 PL=0
MOVL C00443 V=800.0 PL=0
MOVL C00444 V=800.0 PL=0
MOVL C00445 V=800.0 PL=0
MOVL C00446 V=800.0 PL=0
MOVL C00447 V=800.0 PL=0
MOVL C00448 V=800.0 PL=0
MOVL C00449 V=800.0 PL=0
MOVL C00450 V=800.0 PL=0
MOVL C00451 V=800.0 PL=0
MOVL C00452 V=800.0 PL=0
MOVL C00453 V=800.0 PL=0
MOVL C00454 V=800.0 PL=0
MOVL C00455 V=800.0 PL=0
MOVL C00456 V=800.0 PL=0
MOVL C00457 V=800.0 PL=0
MOVL C00458 V=800.0 PL=0
MOVL C00459 V=800.0 PL=0
MOVL C00460 V=800.0 PL=0
MOVL C00461 V=800.0 PL=0
MOVL C00462 V=800.0 PL=0
MOVL C00463 V=800.0 PL=0
MOVL C00464 V=800.0 PL=0
MOVL C00465 V=800.0 PL=0
MOVL C00466 V=800.0 PL=0
MOVL C00467 V=800.0 PL=0
MOVL C00468 V=800.0 PL=0
MOVL C00469 V=800.0 PL=0
MOVL C00470 V=800.0 PL=0
MOVL C00471 V=800.0 PL=0
MOVL C00472 V=800.0 PL=0
MOVL C00473 V=800.0 PL=0
MOVL C00474 V=800.0 PL=0
MOVL C00475 V=800.0 PL=0
MOVL C00476 V=800.0 PL=0
MOVL C00477 V=800.0 PL=0
MOVL C00478 V=800.0 PL=0
MOVL C00479 V=800.0 PL=0
MOVL C00480 V=800.0 PL=0
MOVL C00481 V=800.0 PL=0
MOVL C00482 V=800.0 PL=0
MOVL C00483 V=800.0 PL=0
MOVL C00484 V=800.0 PL=0
MOVL C00485 V=800.0 PL=0
MOVL C00486 V=800.0 PL=0
MOVL C00487 V=800.0 PL=0
MOVL C00488 V=800.0 PL=0
MOVL C00489 V=800.0 PL=0
MOVL C00490 V=800.0 PL=0
MOVL C00491 V=800.0 PL=0
MOVL C00492 V=800.0 PL=0
MOVL C00493 V=800.0 PL=0
MOVL C00494 V=800.0 PL=0
MOVL C00495 V=800.0 PL=0
MOVL C00496 V=800.0 PL=0
MOVL C00497 V=800.0 PL=0
MOVL C00498 V=800.0 PL=0
MOVL C00499 V=800.0 PL=0
MOVL C00500 V=800.0 PL=0
MOVL C00501 V=800.0 PL=0
MOVL C00502 V=800.0 PL=0
MOVL C00503 V=800.0 PL=0
MOVL C00504 V=800.0 PL=0
MOVL C00505 V=800.0 PL=0
MOVL C00506 V=800.0 PL=0
MOVL C00507 V=800.0 PL=0
MOVL C00508 V=800.0 PL=0
MOVL C00509 V=800.0 PL=0
MOVL C00510 V=800.0 PL=0
MOVL C00511 V=800.0 PL=0
MOVL C00512 V=800.0 PL=0
MOVL C00513 V=800.0 PL=0
MOVL C00514 V=800.0 PL=0
MOVL C00515 V=800.0 PL=0
MOVL C00516 V=800.0 PL=0
MOVL C00517 V=800.0 PL=0
MOVL C00518 V=800.0 PL=0
MOVL C00519 V=800.0 PL=0
MOVL C00520 V=800.0 PL=0
MOVL C00521 V=800.0 PL=0
MOVL C00522 V=800.0 PL=0
MOVL C00523 V=800.0 PL=0
MOVL C00524 V=800.0 PL=0
MOVL C00525 V=800.0 PL=0
MOVL C00526 V=800.0 PL=0
MOVL C00527 V=800.0 PL=0
MOVL C00528 V=800.0 PL=0
MOVL C00529 V=800.0 PL=0
MOVL C00530 V=800.0 PL=0
MOVL C00531 V=800.0 PL=0
MOVL C00532 V=800.0 PL=0
MOVL C00533 V=800.0 PL=0
MOVL C00534 V=800.0 PL=0
MOVL C00535 V=800.0 PL=0
MOVL C00536 V=800.0 PL=0
MOVL C00537 V=800.0 PL=0
MOVL C00538 V=800.0 PL=0
MOVL C00539 V=800.0 PL=0
MOVL C00540 V=800.0 PL=0
MOVL C00541 V=800.0 PL=0
MOVL C00542 V=800.0 PL=0
MOVL C00543 V=800.0 PL=0
MOVL C00544 V=800.0 PL=0
MOVL C00545 V=800.0 PL=0
MOVL C00546 V=800.0 PL=0
MOVL C00547 V=800.0 PL=0
MOVL C00548 V=800.0 PL=0
MOVL C00549 V=800.0 PL=0
MOVL C00550 V=800.0 PL=0
MOVL C00551 V=800.0 PL=0
MOVL C00552 V=800.0 PL=0
MOVL C00553 V=800.0 PL=0
MOVL C00554 V=800.0 PL=0
MOVL C00555 V=800.0 PL=0
MOVL C00556 V=800.0 PL=0
MOVL C00557 V=800.0 PL=0
MOVL C00558 V=800.0 PL=0
MOVL C00559 V=800.0 PL=0
MOVL C00560 V=800.0 PL=0
MOVL C00561 V=800.0 PL=0
MOVL C00562 V=800.0 PL=0
MOVL C00563 V=800.0 PL=0
MOVL C00564 V=800.0 PL=0
MOVL C00565 V=800.0 PL=0
MOVL C00566 V=800.0 PL=0
MOVL C00567 V=800.0 PL=0
MOVL C00568 V=800.0 PL=0
MOVL C00569 V=800.0 PL=0
MOVL C00570 V=800.0 PL=0
MOVL C00571 V=800.0 PL=0
MOVL C00572 V=800.0 PL=0
MOVL C00573 V=800.0 PL=0
MOVL C00574 V=800.0 PL=0
MOVL C00575 V=800.0 PL=0
MOVL C00576 V=800.0 PL=0
MOVL C00577 V=800.0 PL=0
MOVL C00578 V=800.0 PL=0
MOVL C00579 V=800.0 PL=0
MOVL C00580 V=800.0 PL=0
MOVL C00581 V=800.0 PL=0
MOVL C00582 V=800.0 PL=0
MOVL C00583 V=800.0 PL=0
MOVL C00584 V=800.0 PL=0
MOVL C00585 V=800.0 PL=0
MOVL C00586 V=800.0 PL=0
MOVL C00587 V=800.0 PL=0
MOVL C00588 V=800.0 PL=0
MOVL C00589 V=800.0 PL=0
MOVL C00590 V=800.0 PL=0
MOVL C00591 V=800.0 PL=0
MOVL C00592 V=800.0 PL=0
MOVL C00593 V=800.0 PL=0
MOVL C00594 V=800.0 PL=0
MOVL C00595 V=800.0 PL=0
MOVL C00596 V=800.0 PL=0
MOVL C00597 V=800.0 PL=0
MOVL C00598 V=800.0 PL=0
MOVL C00599 V=800.0 PL=0
MOVL C00600 V=800.0 PL=0
MOVL C00601 V=800.0 PL=0
MOVL C00602 V=800.0 PL=0
MOVL C00603 V=800.0 PL=0
MOVL C00604 V=800.0 PL=0
MOVL C00605 V=800.0 PL=0
MOVL C00606 V=800.0 PL=0
MOVL C00607 V=800.0 PL=0
MOVL C00608 V=800.0 PL=0
MOVL C00609 V=800.0 PL=0
MOVL C00610 V=800.0 PL=0
MOVL C00611 V=800.0 PL=0
MOVL C00612 V=800.0 PL=0
MOVL C00613 V=800.0 PL=0
MOVL C00614 V=800.0 PL=0
MOVL C00615 V=800.0 PL=0
MOVL C00616 V=800.0 PL=0
MOVL C00617 V=800.0 PL=0
MOVL C00618 V=800.0 PL=0
MOVL C00619 V=800.0 PL=0
MOVL C00620 V=800.0 PL=0
MOVL C00621 V=800.0 PL=0
MOVL C00622 V=800.0 PL=0
MOVL C00623 V=800.0 PL=0
MOVL C00624 V=800.0 PL=0
MOVL C00625 V=800.0 PL=0
MOVL C00626 V=800.0 PL=0
MOVL C00627 V=800.0 PL=0
MOVL C00628 V=800.0 PL=0
MOVL C00629 V=800.0 PL=0
MOVL C00630 V=800.0 PL=0
MOVL C00631 V=800.0 PL=0
MOVL C00632 V=800.0 PL=0
MOVL C00633 V=800.0 PL=0
MOVL C00634 V=800.0 PL=0
MOVL C00635 V=800.0 PL=0
MOVL C00636 V=800.0 PL=0
MOVL C00637 V=800.0 PL=0
MOVL C00638 V=800.0 PL=0
MOVL C00639 V=800.0 PL=0
MOVL C00640 V=800.0 PL=0
MOVL C00641 V=800.0 PL=0
MOVL C00642 V=800.0 PL=0
MOVL C00643 V=800.0 PL=0
MOVL C00644 V=800.0 PL=0
MOVL C00645 V=800.0 PL=0
MOVL C00646 V=800.0 PL=0
MOVL C00647 V=800.0 PL=0
MOVL C00648 V=800.0 PL=0
MOVL C00649 V=800.0 PL=0
MOVL C00650 V=800.0 PL=0
MOVL C00651 V=800.0 PL=0
MOVL C00652 V=800.0 PL=0
MOVL C00653 V=800.0 PL=0
MOVL C00654 V=800.0 PL=0
MOVL C00655 V=800.0 PL=0
MOVL C00656 V=800.0 PL=0
MOVL C00657 V=800.0 PL=0
MOVL C00658 V=800.0 PL=0
MOVL C00659 V=800.0 PL=0
MOVL C00660 V=800.0 PL=0
MOVL C00661 V=800.0 PL=0
MOVL C00662 V=800.0 PL=0
MOVL C00663 V=800.0 PL=0
MOVL C00664 V=800.0 PL=0
MOVL C00665 V=800.0 PL=0
MOVL C00666 V=800.0 PL=0
MOVL C00667 V=800.0 PL=0
MOVL C00668 V=800.0 PL=0
MOVL C00669 V=800.0 PL=0
MOVL C00670 V=800.0 PL=0
MOVL C00671 V=800.0 PL=0
MOVL C00672 V=800.0 PL=0
MOVL C00673 V=800.0 PL=0
MOVL C00674 V=800.0 PL=0
MOVL C00675 V=800.0 PL=0
MOVL C00676 V=800.0 PL=0
MOVL C00677 V=800.0 PL=0
MOVL C00678 V=800.0 PL=0
MOVL C00679 V=800.0 PL=0
MOVL C00680 V=800.0 PL=0
MOVL C00681 V=800.0 PL=0
MOVL C00682 V=800.0 PL=0
MOVL C00683 V=800.0 PL=0
MOVL C00684 V=800.0 PL=0
MOVL C00685 V=800.0 PL=0
MOVL C00686 V=800.0 PL=0
MOVL C00687 V=800.0 PL=0
MOVL C00688 V=800.0 PL=0
MOVL C00689 V=800.0 PL=0
MOVL C00690 V=800.0 PL=0
MOVL C00691 V=800.0 PL=0
MOVL C00692 V=800.0 PL=0
MOVL C00693 V=800.0 PL=0
MOVL C00694 V=800.0 PL=0
MOVL C00695 V=800.0 PL=0
MOVL C00696 V=800.0 PL=0
MOVL C00697 V=800.0 PL=0
MOVL C00698 V=800.0 PL=0
MOVL C00699 V=800.0 PL=0
MOVL C00700 V=800.0 PL=0
MOVL C00701 V=800.0 PL=0
MOVL C00702 V=800.0 PL=0
MOVL C00703 V=800.0 PL=0
MOVL C00704 V=800.0 PL=0
MOVL C00705 V=800.0 PL=0
MOVL C00706 V=800.0 PL=0
MOVL C00707 V=800.0 PL=0
MOVL C00708 V=800.0 PL=0
MOVL C00709 V=800.0 PL=0
MOVL C00710 V=800.0 PL=0
MOVL C00711 V=800.0 PL=0
MOVL C00712 V=800.0 PL=0
MOVL C00713 V=800.0 PL=0
MOVL C00714 V=800.0 PL=0
MOVL C00715 V=800.0 PL=0
MOVL C00716 V=800.0 PL=0
MOVL C00717 V=800.0 PL=0
MOVL C00718 V=800.0 PL=0
MOVL C00719 V=800.0 PL=0
MOVL C00720 V=800.0 PL=0
MOVL C00721 V=800.0 PL=0
MOVL C00722 V=800.0 PL=0
MOVL C00723 V=800.0 PL=0
MOVL C00724 V=800.0 PL=0
MOVL C00725 V=800.0 PL=0
MOVL C00726 V=800.0 PL=0
MOVL C00727 V=800.0 PL=0
MOVL C00728 V=800.0 PL=0
MOVL C00729 V=800.0 PL=0
MOVL C00730 V=800.0 PL=0
MOVL C00731 V=800.0 PL=0
MOVL C00732 V=800.0 PL=0
MOVL C00733 V=800.0 PL=0
MOVL C00734 V=800.0 PL=0
MOVL C00735 V=800.0 PL=0
MOVL C00736 V=800.0 PL=0
MOVL C00737 V=800.0 PL=0
MOVL C00738 V=800.0 PL=0
MOVL C00739 V=800.0 PL=0
MOVL C00740 V=800.0 PL=0
MOVL C00741 V=800.0 PL=0
MOVL C00742 V=800.0 PL=0
MOVL C00743 V=800.0 PL=0
MOVL C00744 V=800.0 PL=0
MOVL C00745 V=800.0 PL=0
MOVL C00746 V=800.0 PL=0
MOVL C00747 V=800.0 PL=0
MOVL C00748 V=800.0 PL=0
MOVL C00749 V=800.0 PL=0
MOVL C00750 V=800.0 PL=0
MOVL C00751 V=800.0 PL=0
MOVL C00752 V=800.0 PL=0
MOVL C00753 V=800.0 PL=0
MOVL C00754 V=800.0 PL=0
MOVL C00755 V=800.0 PL=0
MOVL C00756 V=800.0 PL=0
MOVL C00757 V=800.0 PL=0
MOVL C00758 V=800.0 PL=0
MOVL C00759 V=800.0 PL=0
MOVL C00760 V=800.0 PL=0
MOVL C00761 V=800.0 PL=0
MOVL C00762 V=800.0 PL=0
MOVL C00763 V=800.0 PL=0
MOVL C00764 V=800.0 PL=0
MOVL C00765 V=800.0 PL=0
MOVL C00766 V=800.0 PL=0
MOVL C00767 V=800.0 PL=0
MOVL C00768 V=800.0 PL=0
MOVL C00769 V=800.0 PL=0
MOVL C00770 V=800.0 PL=0
MOVL C00771 V=800.0 PL=0
MOVL C00772 V=800.0 PL=0
MOVL C00773 V=800.0 PL=0
MOVL C00774 V=800.0 PL=0
MOVL C00775 V=800.0 PL=0
MOVL C00776 V=800.0 PL=0
MOVL C00777 V=800.0 PL=0
MOVL C00778 V=800.0 PL=0
MOVL C00779 V=800.0 PL=0
MOVL C00780 V=800.0 PL=0
MOVL C00781 V=800.0 PL=0
MOVL C00782 V=800.0 PL=0
MOVL C00783 V=800.0 PL=0
MOVL C00784 V=800.0 PL=0
MOVL C00785 V=800.0 PL=0
MOVL C00786 V=800.0 PL=0
MOVL C00787 V=800.0 PL=0
MOVL C00788 V=800.0 PL=0
MOVL C00789 V=800.0 PL=0
MOVL C00790 V=800.0 PL=0
MOVL C00791 V=800.0 PL=0
MOVL C00792 V=800.0 PL=0
MOVL C00793 V=800.0 PL=0
MOVL C00794 V=800.0 PL=0
MOVL C00795 V=800.0 PL=0
MOVL C00796 V=800.0 PL=0
MOVL C00797 V=800.0 PL=0
MOVL C00798 V=800.0 PL=0
MOVL C00799 V=800.0 PL=0
MOVL C00800 V=800.0 PL=0
MOVL C00801 V=800.0 PL=0
MOVL C00802 V=800.0 PL=0
MOVL C00803 V=800.0 PL=0
MOVL C00804 V=800.0 PL=0
MOVL C00805 V=800.0 PL=0
MOVL C00806 V=800.0 PL=0
MOVL C00807 V=800.0 PL=0
MOVL C00808 V=800.0 PL=0
MOVL C00809 V=800.0 PL=0
MOVL C00810 V=800.0 PL=0
MOVL C00811 V=800.0 PL=0
MOVL C00812 V=800.0 PL=0
MOVL C00813 V=800.0 PL=0
MOVL C00814 V=800.0 PL=0
MOVL C00815 V=800.0 PL=0
MOVL C00816 V=800.0 PL=0
MOVL C00817 V=800.0 PL=0
MOVL C00818 V=800.0 PL=0
MOVL C00819 V=800.0 PL=0
MOVL C00820 V=800.0 PL=0
MOVL C00821 V=800.0 PL=0
MOVL C00822 V=800.0 PL=0
MOVL C00823 V=800.0 PL=0
MOVL C00824 V=800.0 PL=0
MOVL C00825 V=800.0 PL=0
MOVL C00826 V=800.0 PL=0
MOVL C00827 V=800.0 PL=0
MOVL C00828 V=800.0 PL=0
MOVL C00829 V=800.0 PL=0
MOVL C00830 V=800.0 PL=0
MOVL C00831 V=800.0 PL=0
MOVL C00832 V=800.0 PL=0
MOVL C00833 V=800.0 PL=0
MOVL C00834 V=800.0 PL=0
MOVL C00835 V=800.0 PL=0
MOVL C00836 V=800.0 PL=0
MOVL C00837 V=800.0 PL=0
MOVL C00838 V=800.0 PL=0
MOVL C00839 V=800.0 PL=0
MOVL C00840 V=800.0 PL=0
MOVL C00841 V=800.0 PL=0
MOVL C00842 V=800.0 PL=0
MOVL C00843 V=800.0 PL=0
MOVL C00844 V=800.0 PL=0
MOVL C00845 V=800.0 PL=0
MOVL C00846 V=800.0 PL=0
MOVL C00847 V=800.0 PL=0
MOVL C00848 V=800.0 PL=0
MOVL C00849 V=800.0 PL=0
MOVL C00850 V=800.0 PL=0
MOVL C00851 V=800.0 PL=0
MOVL C00852 V=800.0 PL=0
MOVL C00853 V=800.0 PL=0
MOVL C00854 V=800.0 PL=0
MOVL C00855 V=800.0 PL=0
MOVL C00856 V=800.0 PL=0
MOVL C00857 V=800.0 PL=0
MOVL C00858 V=800.0 PL=0
MOVL C00859 V=800.0 PL=0
MOVL C00860 V=800.0 PL=0
MOVL C00861 V=800.0 PL=0
MOVL C00862 V=800.0 PL=0
MOVL C00863 V=800.0 PL=0
MOVL C00864 V=800.0 PL=0
MOVL C00865 V=800.0 PL=0
MOVL C00866 V=800.0 PL=0
MOVL C00867 V=800.0 PL=0
MOVL C00868 V=800.0 PL=0
MOVL C00869 V=800.0 PL=0
MOVL C00870 V=800.0 PL=0
MOVL C00871 V=800.0 PL=0
MOVL C00872 V=800.0 PL=0
MOVL C00873 V=800.0 PL=0
MOVL C00874 V=800.0 PL=0
MOVL C00875 V=800.0 PL=0
MOVL C00876 V=800.0 PL=0
MOVL C00877 V=800.0 PL=0
MOVL C00878 V=800.0 PL=0
MOVL C00879 V=800.0 PL=0
MOVL C00880 V=800.0 PL=0
MOVL C00881 V=800.0 PL=0
MOVL C00882 V=800.0 PL=0
MOVL C00883 V=800.0 PL=0
MOVL C00884 V=800.0 PL=0
MOVL C00885 V=800.0 PL=0
MOVL C00886 V=800.0 PL=0
MOVL C00887 V=800.0 PL=0
MOVL C00888 V=800.0 PL=0
MOVL C00889 V=800.0 PL=0
MOVL C00890 V=800.0 PL=0
MOVL C00891 V=800.0 PL=0
MOVL C00892 V=800.0 PL=0
MOVL C00893 V=800.0 PL=0
MOVL C00894 V=800.0 PL=0
MOVL C00895 V=800.0 PL=0
MOVL C00896 V=800.0 PL=0
MOVL C00897 V=800.0 PL=0
MOVL C00898 V=800.0 PL=0
MOVL C00899 V=800.0 PL=0
MOVL C00900 V=800.0 PL=0
MOVL C00901 V=800.0 PL=0
MOVL C00902 V=800.0 PL=0
MOVL C00903 V=800.0 PL=0
MOVL C00904 V=800.0 PL=0
MOVL C00905 V=800.0 PL=0
MOVL C00906 V=800.0 PL=0
MOVL C00907 V=800.0 PL=0
MOVL C00908 V=800.0 PL=0
MOVL C00909 V=800.0 PL=0
MOVL C00910 V=800.0 PL=0
MOVL C00911 V=800.0 PL=0
MOVL C00912 V=800.0 PL=0
MOVL C00913 V=800.0 PL=0
MOVL C00914 V=800.0 PL=0
MOVL C00915 V=800.0 PL=0
MOVL C00916 V=800.0 PL=0
MOVL C00917 V=800.0 PL=0
MOVL C00918 V=800.0 PL=0
MOVL C00919 V=800.0 PL=0
MOVL C00920 V=800.0 PL=0
MOVL C00921 V=800.0 PL=0
MOVL C00922 V=800.0 PL=0
MOVL C00923 V=800.0 PL=0
MOVL C00924 V=800.0 PL=0
MOVL C00925 V=800.0 PL=0
MOVL C00926 V=800.0 PL=0
MOVL C00927 V=800.0 PL=0
MOVL C00928 V=800.0 PL=0
MOVL C00929 V=800.0 PL=0
MOVL C00930 V=800.0 PL=0
MOVL C00931 V=800.0 PL=0
MOVL C00932 V=800.0 PL=0
MOVL C00933 V=800.0 PL=0
MOVL C00934 V=800.0 PL=0
MOVL C00935 V=800.0 PL=0
MOVL C00936 V=800.0 PL=0
MOVL C00937 V=800.0 PL=0
MOVL C00938 V=800.0 PL=0
MOVL C00939 V=800.0 PL=0
MOVL C00940 V=800.0 PL=0
MOVL C00941 V=800.0 PL=0
MOVL C00942 V=800.0 PL=0
MOVL C00943 V=800.0 PL=0
MOVL C00944 V=800.0 PL=0
MOVL C00945 V=800.0 PL=0
MOVL C00946 V=800.0 PL=0
MOVL C00947 V=800.0 PL=0
MOVL C00948 V=800.0 PL=0
MOVL C00949 V=800.0 PL=0
MOVL C00950 V=800.0 PL=0
MOVL C00951 V=800.0 PL=0
MOVL C00952 V=800.0 PL=0
MOVL C00953 V=800.0 PL=0
MOVL C00954 V=800.0 PL=0
MOVL C00955 V=800.0 PL=0
MOVL C00956 V=800.0 PL=0
MOVL C00957 V=800.0 PL=0
MOVL C00958 V=800.0 PL=0
MOVL C00959 V=800.0 PL=0
MOVL C00960 V=800.0 PL=0
MOVL C00961 V=800.0 PL=0
MOVL C00962 V=800.0 PL=0
MOVL C00963 V=800.0 PL=0
MOVL C00964 V=800.0 PL=0
MOVL C00965 V=800.0 PL=0
MOVL C00966 V=800.0 PL=0
MOVL C00967 V=800.0 PL=0
MOVL C00968 V=800.0 PL=0
MOVL C00969 V=800.0 PL=0
MOVL C00970 V=800.0 PL=0
MOVL C00971 V=800.0 PL=0
MOVL C00972 V=800.0 PL=0
MOVL C00973 V=800.0 PL=0
MOVL C00974 V=800.0 PL=0
MOVL C00975 V=800.0 PL=0
MOVL C00976 V=800.0 PL=0
MOVL C00977 V=800.0 PL=0
MOVL C00978 V=800.0 PL=0
MOVL C00979 V=800.0 PL=0
MOVL C00980 V=800.0 PL=0
MOVL C00981 V=800.0 PL=0
MOVL C00982 V=800.0 PL=0
MOVL C00983 V=800.0 PL=0
MOVL C00984 V=800.0 PL=0
MOVL C00985 V=800.0 PL=0
MOVL C00986 V=800.0 PL=0
MOVL C00987 V=800.0 PL=0
MOVL C00988 V=800.0 PL=0
MOVL C00989 V=800.0 PL=0
MOVL C00990 V=800.0 PL=0
MOVL C00991 V=800.0 PL=0
MOVL C00992 V=800.0 PL=0
MOVL C00993 V=800.0 PL=0
MOVL C00994 V=800.0 PL=0
MOVL C00995 V=800.0 PL=0
MOVL C00996 V=800.0 PL=0
MOVL C00997 V=800.0 PL=0
MOVL C00998 V=800.0 PL=0
MOVL C00999 V=800.0 PL=0
MOVL C01000 V=800.0 PL=0
MOVL C01001 V=800.0 PL=0
MOVL C01002 V=800.0 PL=0
MOVL C01003 V=800.0 PL=0
MOVL C01004 V=800.0 PL=0
MOVL C01005 V=800.0 PL=0
MOVL C01006 V=800.0 PL=0
MOVL C01007 V=800.0 PL=0
MOVL C01008 V=800.0 PL=0
MOVL C01009 V=800.0 PL=0
MOVL C01010 V=800.0 PL=0
MOVL C01011 V=800.0 PL=0
MOVL C01012 V=800.0 PL=0
MOVL C01013 V=800.0 PL=0
MOVL C01014 V=800.0 PL=0
MOVL C01015 V=800.0 PL=0
MOVL C01016 V=800.0 PL=0
MOVL C01017 V=800.0 PL=0
MOVL C01018 V=800.0 PL=0
MOVL C01019 V=800.0 PL=0
MOVL C01020 V=800.0 PL=0
MOVL C01021 V=800.0 PL=0
MOVL C01022 V=800.0 PL=0
MOVL C01023 V=800.0 PL=0
MOVL C01024 V=800.0 PL=0
MOVL C01025 V=800.0 PL=0
MOVL C01026 V=800.0 PL=0
MOVL C01027 V=800.0 PL=0
MOVL C01028 V=800.0 PL=0
MOVL C01029 V=800.0 PL=0
MOVL C01030 V=800.0 PL=0
MOVL C01031 V=800.0 PL=0
MOVL C01032 V=800.0 PL=0
MOVL C01033 V=800.0 PL=0
MOVL C01034 V=800.0 PL=0
MOVL C01035 V=800.0 PL=0
MOVL C01036 V=800.0 PL=0
MOVL C01037 V=800.0 PL=0
MOVL C01038 V=800.0 PL=0
MOVL C01039 V=800.0 PL=0
MOVL C01040 V=800.0 PL=0
MOVL C01041 V=800.0 PL=0
MOVL C01042 V=800.0 PL=0
MOVL C01043 V=800.0 PL=0
MOVL C01044 V=800.0 PL=0
MOVL C01045 V=800.0 PL=0
MOVL C01046 V=800.0 PL=0
MOVL C01047 V=800.0 PL=0
MOVL C01048 V=800.0 PL=0
MOVL C01049 V=800.0 PL=0
MOVL C01050 V=800.0 PL=0
MOVL C01051 V=800.0 PL=0
MOVL C01052 V=800.0 PL=0
MOVL C01053 V=800.0 PL=0
MOVL C01054 V=800.0 PL=0
MOVL C01055 V=800.0 PL=0
MOVL C01056 V=800.0 PL=0
MOVL C01057 V=800.0 PL=0
MOVL C01058 V=800.0 PL=0
MOVL C01059 V=800.0 PL=0
MOVL C01060 V=800.0 PL=0
MOVL C01061 V=800.0 PL=0
MOVL C01062 V=800.0 PL=0
MOVL C01063 V=800.0 PL=0
MOVL C01064 V=800.0 PL=0
MOVL C01065 V=800.0 PL=0
MOVL C01066 V=800.0 PL=0
MOVL C01067 V=800.0 PL=0
MOVL C01068 V=800.0 PL=0
MOVL C01069 V=800.0 PL=0
MOVL C01070 V=800.0 PL=0
MOVL C01071 V=800.0 PL=0
MOVL C01072 V=800.0 PL=0
MOVL C01073 V=800.0 PL=0
MOVL C01074 V=800.0 PL=0
MOVL C01075 V=800.0 PL=0
MOVL C01076 V=800.0 PL=0
MOVL C01077 V=800.0 PL=0
MOVL C01078 V=800.0 PL=0
MOVL C01079 V=800.0 PL=0
MOVL C01080 V=800.0 PL=0
MOVL C01081 V=800.0 PL=0
MOVL C01082 V=800.0 PL=0
MOVL C01083 V=800.0 PL=0
MOVL C01084 V=800.0 PL=0
MOVL C01085 V=800.0 PL=0
MOVL C01086 V=800.0 PL=0
MOVL C01087 V=800.0 PL=0
MOVL C01088 V=800.0 PL=0
MOVL C01089 V=800.0 PL=0
MOVL C01090 V=800.0 PL=0
MOVL C01091 V=800.0 PL=0
MOVL C01092 V=800.0 PL=0
MOVL C01093 V=800.0 PL=0
MOVL C01094 V=800.0 PL=0
MOVL C01095 V=800.0 PL=0
MOVL C01096 V=800.0 PL=0
MOVL C01097 V=800.0 PL=0
MOVL C01098 V=800.0 PL=0
MOVL C01099 V=800.0 PL=0
MOVL C01100 V=800.0 PL=0
MOVL C01101 V=800.0 PL=0
MOVL C01102 V=800.0 PL=0
MOVL C01103 V=800.0 PL=0
MOVL C01104 V=800.0 PL=0
MOVL C01105 V=800.0 PL=0
MOVL C01106 V=800.0 PL=0
MOVL C01107 V=800.0 PL=0
MOVL C01108 V=800.0 PL=0
MOVL C01109 V=800.0 PL=0
MOVL C01110 V=800.0 PL=0
MOVL C01111 V=800.0 PL=0
MOVL C01112 V=800.0 PL=0
MOVL C01113 V=800.0 PL=0
MOVL C01114 V=800.0 PL=0
MOVL C01115 V=800.0 PL=0
MOVL C01116 V=800.0 PL=0
MOVL C01117 V=800.0 PL=0
MOVL C01118 V=800.0 PL=0
MOVL C01119 V=800.0 PL=0
MOVL C01120 V=800.0 PL=0
MOVL C01121 V=800.0 PL=0
MOVL C01122 V=800.0 PL=0
MOVL C01123 V=800.0 PL=0
MOVL C01124 V=800.0 PL=0
MOVL C01125 V=800.0 PL=0
MOVL C01126 V=800.0 PL=0
MOVL C01127 V=800.0 PL=0
MOVL C01128 V=800.0 PL=0
MOVL C01129 V=800.0 PL=0
MOVL C01130 V=800.0 PL=0
MOVL C01131 V=800.0 PL=0
MOVL C01132 V=800.0 PL=0
MOVL C01133 V=800.0 PL=0
MOVL C01134 V=800.0 PL=0
MOVL C01135 V=800.0 PL=0
MOVL C01136 V=800.0 PL=0
MOVL C01137 V=800.0 PL=0
MOVL C01138 V=800.0 PL=0
MOVL C01139 V=800.0 PL=0
MOVL C01140 V=800.0 PL=0
MOVL C01141 V=800.0 PL=0
MOVL C01142 V=800.0 PL=0
MOVL C01143 V=800.0 PL=0
MOVL C01144 V=800.0 PL=0
MOVL C01145 V=800.0 PL=0
MOVL C01146 V=800.0 PL=0
MOVL C01147 V=800.0 PL=0
MOVL C01148 V=800.0 PL=0
MOVL C01149 V=800.0 PL=0
MOVL C01150 V=800.0 PL=0
MOVL C01151 V=800.0 PL=0
MOVL C01152 V=800.0 PL=0
MOVL C01153 V=800.0 PL=0
MOVL C01154 V=800.0 PL=0
MOVL C01155 V=800.0 PL=0
MOVL C01156 V=800.0 PL=0
MOVL C01157 V=800.0 PL=0
MOVL C01158 V=800.0 PL=0
MOVL C01159 V=800.0 PL=0
MOVL C01160 V=800.0 PL=0
MOVL C01161 V=800.0 PL=0
MOVL C01162 V=800.0 PL=0
MOVL C01163 V=800.0 PL=0
MOVL C01164 V=800.0 PL=0
MOVL C01165 V=800.0 PL=0
MOVL C01166 V=800.0 PL=0
MOVL C01167 V=800.0 PL=0
MOVL C01168 V=800.0 PL=0
MOVL C01169 V=800.0 PL=0
MOVL C01170 V=800.0 PL=0
MOVL C01171 V=800.0 PL=0
MOVL C01172 V=800.0 PL=0
MOVL C01173 V=800.0 PL=0
MOVL C01174 V=800.0 PL=0
MOVL C01175 V=800.0 PL=0
MOVL C01176 V=800.0 PL=0
MOVL C01177 V=800.0 PL=0
MOVL C01178 V=800.0 PL=0
MOVL C01179 V=800.0 PL=0
MOVL C01180 V=800.0 PL=0
MOVL C01181 V=800.0 PL=0
MOVL C01182 V=800.0 PL=0
MOVL C01183 V=800.0 PL=0
MOVL C01184 V=800.0 PL=0
MOVL C01185 V=800.0 PL=0
MOVL C01186 V=800.0 PL=0
MOVL C01187 V=800.0 PL=0
MOVL C01188 V=800.0 PL=0
MOVL C01189 V=800.0 PL=0
MOVL C01190 V=800.0 PL=0
MOVL C01191 V=800.0 PL=0
MOVL C01192 V=800.0 PL=0
MOVL C01193 V=800.0 PL=0
MOVL C01194 V=800.0 PL=0
MOVL C01195 V=800.0 PL=0
MOVL C01196 V=800.0 PL=0
MOVL C01197 V=800.0 PL=0
MOVL C01198 V=800.0 PL=0
MOVL C01199 V=800.0 PL=0
MOVL C01200 V=800.0 PL=0
MOVL C01201 V=800.0 PL=0
MOVL C01202 V=800.0 PL=0
MOVL C01203 V=800.0 PL=0
MOVL C01204 V=800.0 PL=0
MOVL C01205 V=800.0 PL=0
MOVL C01206 V=800.0 PL=0
MOVL C01207 V=800.0 PL=0
MOVL C01208 V=800.0 PL=0
MOVL C01209 V=800.0 PL=0
MOVL C01210 V=800.0 PL=0
MOVL C01211 V=800.0 PL=0
MOVL C01212 V=800.0 PL=0
MOVL C01213 V=800.0 PL=0
MOVL C01214 V=800.0 PL=0
MOVL C01215 V=800.0 PL=0
MOVL C01216 V=800.0 PL=0
MOVL C01217 V=800.0 PL=0
MOVL C01218 V=800.0 PL=0
MOVL C01219 V=800.0 PL=0
MOVL C01220 V=800.0 PL=0
MOVL C01221 V=800.0 PL=0
MOVL C01222 V=800.0 PL=0
MOVL C01223 V=800.0 PL=0
MOVL C01224 V=800.0 PL=0
MOVL C01225 V=800.0 PL=0
MOVL C01226 V=800.0 PL=0
MOVL C01227 V=800.0 PL=0
MOVL C01228 V=800.0 PL=0
MOVL C01229 V=800.0 PL=0
MOVL C01230 V=800.0 PL=0
MOVL C01231 V=800.0 PL=0
MOVL C01232 V=800.0 PL=0
MOVL C01233 V=800.0 PL=0
MOVL C01234 V=800.0 PL=0
MOVL C01235 V=800.0 PL=0
MOVL C01236 V=800.0 PL=0
MOVL C01237 V=800.0 PL=0
MOVL C01238 V=800.0 PL=0
MOVL C01239 V=800.0 PL=0
MOVL C01240 V=800.0 PL=0
MOVL C01241 V=800.0 PL=0
MOVL C01242 V=800.0 PL=0
MOVL C01243 V=800.0 PL=0
MOVL C01244 V=800.0 PL=0
MOVL C01245 V=800.0 PL=0
MOVL C01246 V=800.0 PL=0
MOVL C01247 V=800.0 PL=0
MOVL C01248 V=800.0 PL=0
MOVL C01249 V=800.0 PL=0
MOVL C01250 V=800.0 PL=0
MOVL C01251 V=800.0 PL=0
MOVL C01252 V=800.0 PL=0
MOVL C01253 V=800.0 PL=0
MOVL C01254 V=800.0 PL=0
MOVL C01255 V=800.0 PL=0
MOVL C01256 V=800.0 PL=0
MOVL C01257 V=800.0 PL=0
MOVL C01258 V=800.0 PL=0
MOVL C01259 V=800.0 PL=0
MOVL C01260 V=800.0 PL=0
MOVL C01261 V=800.0 PL=0
MOVL C01262 V=800.0 PL=0
MOVL C01263 V=800.0 PL=0
MOVL C01264 V=800.0 PL=0
MOVL C01265 V=800.0 PL=0
MOVL C01266 V=800.0 PL=0
MOVL C01267 V=800.0 PL=0
MOVL C01268 V=800.0 PL=0
MOVL C01269 V=800.0 PL=0
MOVL C01270 V=800.0 PL=0
MOVL C01271 V=800.0 PL=0
MOVL C01272 V=800.0 PL=0
MOVL C01273 V=800.0 PL=0
MOVL C01274 V=800.0 PL=0
MOVL C01275 V=800.0 PL=0
MOVL C01276 V=800.0 PL=0
MOVL C01277 V=800.0 PL=0
MOVL C01278 V=800.0 PL=0
MOVL C01279 V=800.0 PL=0
MOVL C01280 V=800.0 PL=0
MOVL C01281 V=800.0 PL=0
MOVL C01282 V=800.0 PL=0
MOVL C01283 V=800.0 PL=0
MOVL C01284 V=800.0 PL=0
MOVL C01285 V=800.0 PL=0
MOVL C01286 V=800.0 PL=0
MOVL C01287 V=800.0 PL=0
MOVL C01288 V=800.0 PL=0
MOVL C01289 V=800.0 PL=0
MOVL C01290 V=800.0 PL=0
MOVL C01291 V=800.0 PL=0
MOVL C01292 V=800.0 PL=0
MOVL C01293 V=800.0 PL=0
MOVL C01294 V=800.0 PL=0
MOVL C01295 V=800.0 PL=0
MOVL C01296 V=800.0 PL=0
MOVL C01297 V=800.0 PL=0
MOVL C01298 V=800.0 PL=0
MOVL C01299 V=800.0 PL=0
MOVL C01300 V=800.0 PL=0
MOVL C01301 V=800.0 PL=0
MOVL C01302 V=800.0 PL=0
MOVL C01303 V=800.0 PL=0
MOVL C01304 V=800.0 PL=0
MOVL C01305 V=800.0 PL=0
MOVL C01306 V=800.0 PL=0
MOVL C01307 V=800.0 PL=0
MOVL C01308 V=800.0 PL=0
MOVL C01309 V=800.0 PL=0
MOVL C01310 V=800.0 PL=0
MOVL C01311 V=800.0 PL=0
MOVL C01312 V=800.0 PL=0
MOVL C01313 V=800.0 PL=0
MOVL C01314 V=800.0 PL=0
MOVL C01315 V=800.0 PL=0
MOVL C01316 V=800.0 PL=0
MOVL C01317 V=800.0 PL=0
MOVL C01318 V=800.0 PL=0
MOVL C01319 V=800.0 PL=0
MOVL C01320 V=800.0 PL=0
MOVL C01321 V=800.0 PL=0
MOVL C01322 V=800.0 PL=0
MOVL C01323 V=800.0 PL=0
MOVL C01324 V=800.0 PL=0
MOVL C01325 V=800.0 PL=0
MOVL C01326 V=800.0 PL=0
MOVL C01327 V=800.0 PL=0
MOVL C01328 V=800.0 PL=0
MOVL C01329 V=800.0 PL=0
MOVL C01330 V=800.0 PL=0
MOVL C01331 V=800.0 PL=0
MOVL C01332 V=800.0 PL=0
MOVL C01333 V=800.0 PL=0
MOVL C01334 V=800.0 PL=0
MOVL C01335 V=800.0 PL=0
MOVL C01336 V=800.0 PL=0
MOVL C01337 V=800.0 PL=0
MOVL C01338 V=800.0 PL=0
MOVL C01339 V=800.0 PL=0
MOVL C01340 V=800.0 PL=0
MOVL C01341 V=800.0 PL=0
MOVL C01342 V=800.0 PL=0
MOVL C01343 V=800.0 PL=0
MOVL C01344 V=800.0 PL=0
MOVL C01345 V=800.0 PL=0
MOVL C01346 V=800.0 PL=0
MOVL C01347 V=800.0 PL=0
MOVL C01348 V=800.0 PL=0
MOVL C01349 V=800.0 PL=0
MOVL C01350 V=800.0 PL=0
MOVL C01351 V=800.0 PL=0
MOVL C01352 V=800.0 PL=0
MOVL C01353 V=800.0 PL=0
MOVL C01354 V=800.0 PL=0
MOVL C01355 V=800.0 PL=0
MOVL C01356 V=800.0 PL=0
MOVL C01357 V=800.0 PL=0
MOVL C01358 V=800.0 PL=0
MOVL C01359 V=800.0 PL=0
MOVL C01360 V=800.0 PL=0
MOVL C01361 V=800.0 PL=0
MOVL C01362 V=800.0 PL=0
MOVL C01363 V=800.0 PL=0
MOVL C01364 V=800.0 PL=0
MOVL C01365 V=800.0 PL=0
MOVL C01366 V=800.0 PL=0
MOVL C01367 V=800.0 PL=0
MOVL C01368 V=800.0 PL=0
MOVL C01369 V=800.0 PL=0
MOVL C01370 V=800.0 PL=0
MOVL C01371 V=800.0 PL=0
MOVL C01372 V=800.0 PL=0
MOVL C01373 V=800.0 PL=0
MOVL C01374 V=800.0 PL=0
MOVL C01375 V=800.0 PL=0
MOVL C01376 V=800.0 PL=0
MOVL C01377 V=800.0 PL=0
MOVL C01378 V=800.0 PL=0
MOVL C01379 V=800.0 PL=0
MOVL C01380 V=800.0 PL=0
MOVL C01381 V=800.0 PL=0
MOVL C01382 V=800.0 PL=0
MOVL C01383 V=800.0 PL=0
MOVL C01384 V=800.0 PL=0
MOVL C01385 V=800.0 PL=0
MOVL C01386 V=800.0 PL=0
MOVL C01387 V=800.0 PL=0
MOVL C01388 V=800.0 PL=0
MOVL C01389 V=800.0 PL=0
MOVL C01390 V=800.0 PL=0
MOVL C01391 V=800.0 PL=0
MOVL C01392 V=800.0 PL=0
MOVL C01393 V=800.0 PL=0
MOVL C01394 V=800.0 PL=0
MOVL C01395 V=800.0 PL=0
MOVL C01396 V=800.0 PL=0
MOVL C01397 V=800.0 PL=0
MOVL C01398 V=800.0 PL=0
MOVL C01399 V=800.0 PL=0
MOVL C01400 V=800.0 PL=0
MOVL C01401 V=800.0 PL=0
MOVL C01402 V=800.0 PL=0
MOVL C01403 V=800.0 PL=0
MOVL C01404 V=800.0 PL=0
MOVL C01405 V=800.0 PL=0
MOVL C01406 V=800.0 PL=0
MOVL C01407 V=800.0 PL=0
MOVL C01408 V=800.0 PL=0
MOVL C01409 V=800.0 PL=0
MOVL C01410 V=800.0 PL=0
MOVL C01411 V=800.0 PL=0
MOVL C01412 V=800.0 PL=0
MOVL C01413 V=800.0 PL=0
MOVL C01414 V=800.0 PL=0
MOVL C01415 V=800.0 PL=0
MOVL C01416 V=800.0 PL=0
MOVL C01417 V=800.0 PL=0
MOVL C01418 V=800.0 PL=0
MOVL C01419 V=800.0 PL=0
MOVL C01420 V=800.0 PL=0
MOVL C01421 V=800.0 PL=0
MOVL C01422 V=800.0 PL=0
MOVL C01423 V=800.0 PL=0
MOVL C01424 V=800.0 PL=0
MOVL C01425 V=800.0 PL=0
MOVL C01426 V=800.0 PL=0
MOVL C01427 V=800.0 PL=0
MOVL C01428 V=800.0 PL=0
MOVL C01429 V=800.0 PL=0
MOVL C01430 V=800.0 PL=0
MOVL C01431 V=800.0 PL=0
MOVL C01432 V=800.0 PL=0
MOVL C01433 V=800.0 PL=0
MOVL C01434 V=800.0 PL=0
MOVL C01435 V=800.0 PL=0
MOVL C01436 V=800.0 PL=0
MOVL C01437 V=800.0 PL=0
MOVL C01438 V=800.0 PL=0
MOVL C01439 V=800.0 PL=0
MOVL C01440 V=800.0 PL=0
MOVL C01441 V=800.0 PL=0
MOVL C01442 V=800.0 PL=0
MOVL C01443 V=800.0 PL=0
MOVL C01444 V=800.0 PL=0
MOVL C01445 V=800.0 PL=0
MOVL C01446 V=800.0 PL=0
MOVL C01447 V=800.0 PL=0
MOVL C01448 V=800.0 PL=0
MOVL C01449 V=800.0 PL=0
MOVL C01450 V=800.0 PL=0
MOVL C01451 V=800.0 PL=0
MOVL C01452 V=800.0 PL=0
MOVL C01453 V=800.0 PL=0
MOVL C01454 V=800.0 PL=0
MOVL C01455 V=800.0 PL=0
MOVL C01456 V=800.0 PL=0
MOVL C01457 V=800.0 PL=0
MOVL C01458 V=800.0 PL=0
MOVL C01459 V=800.0 PL=0
MOVL C01460 V=800.0 PL=0
MOVL C01461 V=800.0 PL=0
MOVL C01462 V=800.0 PL=0
MOVL C01463 V=800.0 PL=0
MOVL C01464 V=800.0 PL=0
MOVL C01465 V=800.0 PL=0
MOVL C01466 V=800.0 PL=0
MOVL C01467 V=800.0 PL=0
MOVL C01468 V=800.0 PL=0
MOVL C01469 V=800.0 PL=0
MOVL C01470 V=800.0 PL=0
MOVL C01471 V=800.0 PL=0
MOVL C01472 V=800.0 PL=0
MOVL C01473 V=800.0 PL=0
MOVL C01474 V=800.0 PL=0
MOVL C01475 V=800.0 PL=0
MOVL C01476 V=800.0 PL=0
MOVL C01477 V=800.0 PL=0
MOVL C01478 V=800.0 PL=0
MOVL C01479 V=800.0 PL=0
MOVL C01480 V=800.0 PL=0
MOVL C01481 V=800.0 PL=0
MOVL C01482 V=800.0 PL=0
MOVL C01483 V=800.0 PL=0
MOVL C01484 V=800.0 PL=0
MOVL C01485 V=800.0 PL=0
MOVL C01486 V=800.0 PL=0
MOVL C01487 V=800.0 PL=0
MOVL C01488 V=800.0 PL=0
MOVL C01489 V=800.0 PL=0
MOVL C01490 V=800.0 PL=0
MOVL C01491 V=800.0 PL=0
MOVL C01492 V=800.0 PL=0
MOVL C01493 V=800.0 PL=0
MOVL C01494 V=800.0 PL=0
MOVL C01495 V=800.0 PL=0
MOVL C01496 V=800.0 PL=0
MOVL C01497 V=800.0 PL=0
MOVL C01498 V=800.0 PL=0
MOVL C01499 V=800.0 PL=0
MOVL C01500 V=800.0 PL=0
MOVL C01501 V=800.0 PL=0
MOVL C01502 V=800.0 PL=0
MOVL C01503 V=800.0 PL=0
MOVL C01504 V=800.0 PL=0
MOVL C01505 V=800.0 PL=0
MOVL C01506 V=800.0 PL=0
MOVL C01507 V=800.0 PL=0
MOVL C01508 V=800.0 PL=0
MOVL C01509 V=800.0 PL=0
MOVL C01510 V=800.0 PL=0
MOVL C01511 V=800.0 PL=0
MOVL C01512 V=800.0 PL=0
MOVL C01513 V=800.0 PL=0
MOVL C01514 V=800.0 PL=0
MOVL C01515 V=800.0 PL=0
MOVL C01516 V=800.0 PL=0
MOVL C01517 V=800.0 PL=0
MOVL C01518 V=800.0 PL=0
MOVL C01519 V=800.0 PL=0
MOVL C01520 V=800.0 PL=0
MOVL C01521 V=800.0 PL=0
MOVL C01522 V=800.0 PL=0
MOVL C01523 V=800.0 PL=0
MOVL C01524 V=800.0 PL=0
MOVL C01525 V=800.0 PL=0
MOVL C01526 V=800.0 PL=0
MOVL C01527 V=800.0 PL=0
MOVL C01528 V=800.0 PL=0
MOVL C01529 V=800.0 PL=0
MOVL C01530 V=800.0 PL=0
MOVL C01531 V=800.0 PL=0
MOVL C01532 V=800.0 PL=0
MOVL C01533 V=800.0 PL=0
MOVL C01534 V=800.0 PL=0
MOVL C01535 V=800.0 PL=0
MOVL C01536 V=800.0 PL=0
MOVL C01537 V=800.0 PL=0
MOVL C01538 V=800.0 PL=0
MOVL C01539 V=800.0 PL=0
MOVL C01540 V=800.0 PL=0
MOVL C01541 V=800.0 PL=0
MOVL C01542 V=800.0 PL=0
MOVL C01543 V=800.0 PL=0
MOVL C01544 V=800.0 PL=0
MOVL C01545 V=800.0 PL=0
MOVL C01546 V=800.0 PL=0
MOVL C01547 V=800.0 PL=0
MOVL C01548 V=800.0 PL=0
MOVL C01549 V=800.0 PL=0
MOVL C01550 V=800.0 PL=0
MOVL C01551 V=800.0 PL=0
MOVL C01552 V=800.0 PL=0
MOVL C01553 V=800.0 PL=0
MOVL C01554 V=800.0 PL=0
MOVL C01555 V=800.0 PL=0
MOVL C01556 V=800.0 PL=0
MOVL C01557 V=800.0 PL=0
MOVL C01558 V=800.0 PL=0
MOVL C01559 V=800.0 PL=0
MOVL C01560 V=800.0 PL=0
MOVL C01561 V=800.0 PL=0
MOVL C01562 V=800.0 PL=0
MOVL C01563 V=800.0 PL=0
MOVL C01564 V=800.0 PL=0
MOVL C01565 V=800.0 PL=0
MOVL C01566 V=800.0 PL=0
MOVL C01567 V=800.0 PL=0
MOVL C01568 V=800.0 PL=0
MOVL C01569 V=800.0 PL=0
MOVL C01570 V=800.0 PL=0
MOVL C01571 V=800.0 PL=0
MOVL C01572 V=800.0 PL=0
MOVL C01573 V=800.0 PL=0
MOVL C01574 V=800.0 PL=0
MOVL C01575 V=800.0 PL=0
MOVL C01576 V=800.0 PL=0
MOVL C01577 V=800.0 PL=0
MOVL C01578 V=800.0 PL=0
MOVL C01579 V=800.0 PL=0
MOVL C01580 V=800.0 PL=0
MOVL C01581 V=800.0 PL=0
MOVL C01582 V=800.0 PL=0
MOVL C01583 V=800.0 PL=0
MOVL C01584 V=800.0 PL=0
MOVL C01585 V=800.0 PL=0
MOVL C01586 V=800.0 PL=0
MOVL C01587 V=800.0 PL=0
MOVL C01588 V=800.0 PL=0
MOVL C01589 V=800.0 PL=0
MOVL C01590 V=800.0 PL=0
MOVL C01591 V=800.0 PL=0
MOVL C01592 V=800.0 PL=0
MOVL C01593 V=800.0 PL=0
MOVL C01594 V=800.0 PL=0
MOVL C01595 V=800.0 PL=0
MOVL C01596 V=800.0 PL=0
MOVL C01597 V=800.0 PL=0
MOVL C01598 V=800.0 PL=0
MOVL C01599 V=800.0 PL=0
MOVL C01600 V=800.0 PL=0
MOVL C01601 V=800.0 PL=0
MOVL C01602 V=800.0 PL=0
MOVL C01603 V=800.0 PL=0
MOVL C01604 V=800.0 PL=0
MOVL C01605 V=800.0 PL=0
MOVL C01606 V=800.0 PL=0
MOVL C01607 V=800.0 PL=0
MOVL C01608 V=800.0 PL=0
MOVL C01609 V=800.0 PL=0
MOVL C01610 V=800.0 PL=0
MOVL C01611 V=800.0 PL=0
MOVL C01612 V=800.0 PL=0
MOVL C01613 V=800.0 PL=0
MOVL C01614 V=800.0 PL=0
MOVL C01615 V=800.0 PL=0
MOVL C01616 V=800.0 PL=0
MOVL C01617 V=800.0 PL=0
MOVL C01618 V=800.0 PL=0
MOVL C01619 V=800.0 PL=0
MOVL C01620 V=800.0 PL=0
MOVL C01621 V=800.0 PL=0
MOVL C01622 V=800.0 PL=0
MOVL C01623 V=800.0 PL=0
MOVL C01624 V=800.0 PL=0
MOVL C01625 V=800.0 PL=0
MOVL C01626 V=800.0 PL=0
MOVL C01627 V=800.0 PL=0
MOVL C01628 V=800.0 PL=0
MOVL C01629 V=800.0 PL=0
MOVL C01630 V=800.0 PL=0
MOVL C01631 V=800.0 PL=0
MOVL C01632 V=800.0 PL=0
MOVL C01633 V=800.0 PL=0
MOVL C01634 V=800.0 PL=0
MOVL C01635 V=800.0 PL=0
MOVL C01636 V=800.0 PL=0
MOVL C01637 V=800.0 PL=0
MOVL C01638 V=800.0 PL=0
MOVL C01639 V=800.0 PL=0
MOVL C01640 V=800.0 PL=0
MOVL C01641 V=800.0 PL=0
MOVL C01642 V=800.0 PL=0
MOVL C01643 V=800.0 PL=0
MOVL C01644 V=800.0 PL=0
MOVL C01645 V=800.0 PL=0
MOVL C01646 V=800.0 PL=0
MOVL C01647 V=800.0 PL=0
MOVL C01648 V=800.0 PL=0
MOVL C01649 V=800.0 PL=0
MOVL C01650 V=800.0 PL=0
MOVL C01651 V=800.0 PL=0
MOVL C01652 V=800.0 PL=0
MOVL C01653 V=800.0 PL=0
MOVL C01654 V=800.0 PL=0
MOVL C01655 V=800.0 PL=0
MOVL C01656 V=800.0 PL=0
MOVL C01657 V=800.0 PL=0
MOVL C01658 V=800.0 PL=0
MOVL C01659 V=800.0 PL=0
MOVL C01660 V=800.0 PL=0
MOVL C01661 V=800.0 PL=0
MOVL C01662 V=800.0 PL=0
MOVL C01663 V=800.0 PL=0
MOVL C01664 V=800.0 PL=0
MOVL C01665 V=800.0 PL=0
MOVL C01666 V=800.0 PL=0
MOVL C01667 V=800.0 PL=0
MOVL C01668 V=800.0 PL=0
MOVL C01669 V=800.0 PL=0
MOVL C01670 V=800.0 PL=0
MOVL C01671 V=800.0 PL=0
MOVL C01672 V=800.0 PL=0
MOVL C01673 V=800.0 PL=0
MOVL C01674 V=800.0 PL=0
MOVL C01675 V=800.0 PL=0
MOVL C01676 V=800.0 PL=0
MOVL C01677 V=800.0 PL=0
MOVL C01678 V=800.0 PL=0
MOVL C01679 V=800.0 PL=0
MOVL C01680 V=800.0 PL=0
MOVL C01681 V=800.0 PL=0
MOVL C01682 V=800.0 PL=0
MOVL C01683 V=800.0 PL=0
MOVL C01684 V=800.0 PL=0
MOVL C01685 V=800.0 PL=0
MOVL C01686 V=800.0 PL=0
MOVL C01687 V=800.0 PL=0
MOVL C01688 V=800.0 PL=0
MOVL C01689 V=800.0 PL=0
MOVL C01690 V=800.0 PL=0
MOVL C01691 V=800.0 PL=0
MOVL C01692 V=800.0 PL=0
MOVL C01693 V=800.0 PL=0
MOVL C01694 V=800.0 PL=0
MOVL C01695 V=800.0 PL=0
MOVL C01696 V=800.0 PL=0
MOVL C01697 V=800.0 PL=0
MOVL C01698 V=800.0 PL=0
MOVL C01699 V=800.0 PL=0
MOVL C01700 V=800.0 PL=0
MOVL C01701 V=800.0 PL=0
MOVL C01702 V=800.0 PL=0
MOVL C01703 V=800.0 PL=0
MOVL C01704 V=800.0 PL=0
MOVL C01705 V=800.0 PL=0
MOVL C01706 V=800.0 PL=0
MOVL C01707 V=800.0 PL=0
MOVL C01708 V=800.0 PL=0
MOVL C01709 V=800.0 PL=0
MOVL C01710 V=800.0 PL=0
MOVL C01711 V=800.0 PL=0
MOVL C01712 V=800.0 PL=0
MOVL C01713 V=800.0 PL=0
MOVL C01714 V=800.0 PL=0
MOVL C01715 V=800.0 PL=0
MOVL C01716 V=800.0 PL=0
MOVL C01717 V=800.0 PL=0
MOVL C01718 V=800.0 PL=0
MOVL C01719 V=800.0 PL=0
MOVL C01720 V=800.0 PL=0
MOVL C01721 V=800.0 PL=0
MOVL C01722 V=800.0 PL=0
MOVL C01723 V=800.0 PL=0
MOVL C01724 V=800.0 PL=0
MOVL C01725 V=800.0 PL=0
MOVL C01726 V=800.0 PL=0
MOVL C01727 V=800.0 PL=0
MOVL C01728 V=800.0 PL=0
MOVL C01729 V=800.0 PL=0
MOVL C01730 V=800.0 PL=0
MOVL C01731 V=800.0 PL=0
MOVL C01732 V=800.0 PL=0
MOVL C01733 V=800.0 PL=0
